(*initialisation de l'opération*)
OP_Purge(
	CTRL_PLC:= CTRL_PLC,
	RESET:= RESET,
	ENABLE_INT:= IN_FE11T AND IN_FE12T AND OP_Test_RP.AR,
	MANUAL:= MANUAL,
	RESTART_ENABLE_IF_OK:= FALSE,
	N_STEP_OP_OK:= 7,
	N_STEP_OP_NOK:=0);

(*appel de l'action de préparation de l'opération*)
OP_Purge.PRL();


(*GRAFCET*)
(* initialisation du grafcet*)
IF 		OP_Purge.Etape = 0
		THEN
				OP_Purge.Etape.0:= TRUE;
(*repositionnement sur étape 0*)
ELSIF	MANUAL OR RESET OR OP_Arret_Pompes.Etape.1
		OR (OP_Isolement.Etape.1 AND NOT OP_Ventilation.Etape.1)
		OR (OP_Pompage_Sec.Etape.1 AND NOT OP_Purge.Etape.6)
		THEN
				OP_Purge.Etape := 0;
				OP_Purge.Etape.0:=TRUE;
(*étape 0-1*)
ELSIF 	OP_Purge.Etape.0
		AND OP_Purge.Marche_OP
		THEN
				OP_Purge.Etape.1:=TRUE;
				OP_Purge.Etape.0:=FALSE;
(*étape 1-2*)
ELSIF	OP_Purge.Etape.1
		AND OP_Pompage_Sec.Etape.0 AND OP_Pompage_Prim.Etape.0 AND OP_Pompage_Proc.Etape.0
		AND OP_Ventilation.Etape.0 AND OP_Isolement.Etape.0
		THEN
				OP_Purge.Etape.2:=TRUE;
				OP_Purge.Etape.1:=FALSE;
(*étape 2-3*)
ELSIF 	OP_Purge.Etape.2
		AND OP_Pompage_Prim.OK AND TH_Vide_Primaire
		THEN
				OP_Purge.Etape.3:=TRUE;
				OP_Purge.Etape.2:=FALSE;
(*étape 3-4*)
ELSIF 	OP_Purge.Etape.3
		AND TIMER_Purge.Q
		THEN
				OP_Purge.Etape.4:=TRUE;
				OP_Purge.Etape.3:=FALSE;
(*étape 3-2*)
ELSIF 	OP_Purge.Etape.3
		AND NOT OP_Pompage_Prim.OK
		THEN
				OP_Purge.Etape.2:=TRUE;
				OP_Purge.Etape.3:=FALSE;
(*étape 4-5*)
ELSIF 	OP_Purge.Etape.4
		AND TH_Atm
		THEN
				OP_Purge.Etape.5:=TRUE;
				OP_Purge.Etape.4:=FALSE;
(*étape 5-2*)
ELSIF 	OP_Purge.Etape.5
		AND (VAR_Iter_Purge < PRM_N_Purge)
		THEN
				OP_Purge.Etape.2:=TRUE;
				OP_Purge.Etape.5:=FALSE;
(*étape 5-6*)
ELSIF 	OP_Purge.Etape.5
		AND (VAR_Iter_Purge >= PRM_N_Purge)
		THEN
				OP_Purge.Etape.6:=TRUE;
				OP_Purge.Etape.5:=FALSE;
(*étape 6-7*)
ELSIF 	OP_Purge.Etape.6
		AND OP_Pompage_Sec.EC
		THEN
				OP_Purge.Etape.7:=TRUE;
				OP_Purge.Etape.6:=FALSE;
END_IF;

(*cloture du traitement de l'opération*)
OP_Purge.POST();
END_ACTION

ACTION ACT_REGEN:
(*OPERATION REGENERATION POMPE CRYOGENIQUE*)
(*isolement pompage et lancement régénération*)

(*initialisation de l'opération*)
OP_Regen(
	CTRL_PLC:= CTRL_PLC,
	RESET:= RESET,
	ENABLE_INT:= OP_Test_RP.AR AND NOT OP_Marche_Pompes.AR,
	MANUAL:= MANUAL,
	RESTART_ENABLE_IF_OK:= FALSE,
	N_STEP_OP_OK:= 6,
	N_STEP_OP_NOK:=0);

(*appel de l'action de préparation de l'opération*)
OP_Regen.PRL();


(*GRAFCET*)
(* initialisation du grafcet*)
IF 		OP_Regen.Etape = 0
		THEN
				OP_Regen.Etape.0:= TRUE;
(*repositionnement sur étape 0*)
ELSIF	MANUAL OR RESET OR OP_Arret_Pompes.Etape.1
		THEN
				OP_Regen.Etape := 0;
				OP_Regen.Etape.0:=TRUE;
(*étape 0-1*)
ELSIF 	OP_Regen.Etape.0
		AND (OP_Regen.Marche_OP OR (FM_REGEN.Q AND NOT MANUAL AND NOT OP_Regen_Part.EC))
		THEN
				OP_Regen.Etape.1:=TRUE;
				OP_Regen.Etape.0:=FALSE;
(*étape 1-2*)
ELSIF	OP_Regen.Etape.1
		THEN
				OP_Regen.Etape.2:=TRUE;
				OP_Regen.Etape.1:=FALSE;
(*étape 2-3*)
ELSIF 	OP_Regen.Etape.2
		AND (OP_Isolement.Etape.4 OR (OP_Pompage_Prim.Etape.0 AND OP_Pompage_Proc.Etape.0 OR OP_Pompage_Sec.Etape.0 OR OP_Purge.Etape.0))
		THEN
				OP_Regen.Etape.3:=TRUE;
				OP_Regen.Etape.2:=FALSE;
(*étape 3-4*)
ELSIF	OP_Regen.Etape.3 AND PS11.STATE_Regen
		THEN
				OP_Regen.Etape.4:=TRUE;
				OP_Regen.Etape.3:=FALSE;
(*étape 4-5*)
ELSIF	OP_Regen.Etape.4 AND NOT PS11.STATE_Regen
		THEN
				OP_Regen.Etape.5:=TRUE;
				OP_Regen.Etape.4:=FALSE;
(*étape 5-6*)
ELSIF	OP_Regen.Etape.5
		AND (OP_Pompage_Sec.OK OR (OP_Marche_Pompes.OK AND (TH_Atm OR NOT OP_Pompage_Sec.ENABLE_INT)))
		THEN
				OP_Regen.Etape.6:=TRUE;
				OP_Regen.Etape.5:=FALSE;
(*étape 6-0*)
ELSIF	OP_Regen.Etape.6
		AND TIMER_etape6_regen.Q
		THEN
				OP_Regen.Etape.0:=TRUE;
				OP_Regen.Etape.6:=FALSE;
END_IF;

(*cloture du traitement de l'opération*)
OP_Regen.POST();
END_ACTION

ACTION ACT_REGEN_PART:
(*OPERATION REGENERATION POMPE CRYOGENIQUE*)
(*isolement pompage et lancement régénération*)

(*initialisation de l'opération*)
OP_Regen_Part(
	CTRL_PLC:= CTRL_PLC,
	RESET:= RESET,
	ENABLE_INT:= OP_Test_RP.AR AND NOT OP_Marche_Pompes.AR,
	MANUAL:= MANUAL,
	RESTART_ENABLE_IF_OK:= FALSE,
	N_STEP_OP_OK:= 6,
	N_STEP_OP_NOK:=0);

(*appel de l'action de préparation de l'opération*)
OP_Regen_Part.PRL();


(*GRAFCET*)
(* initialisation du grafcet*)
IF 		OP_Regen_Part.Etape = 0
		THEN
				OP_Regen_Part.Etape.0:= TRUE;
(*repositionnement sur étape 0*)
ELSIF	MANUAL OR RESET OR OP_Arret_Pompes.Etape.1
		OR OP_Pompage_Sec.Etape.1 OR OP_Pompage_Prim.Etape.1
		THEN
				OP_Regen_Part.Etape := 0;
				OP_Regen_Part.Etape.0:=TRUE;
(*étape 0-1*)
ELSIF 	OP_Regen_Part.Etape.0
		AND OP_Regen_Part.Marche_OP
		THEN
				OP_Regen_Part.Etape.1:=TRUE;
				OP_Regen_Part.Etape.0:=FALSE;
(*étape 1-2*)
ELSIF	OP_Regen_Part.Etape.1
		THEN
				OP_Regen_Part.Etape.2:=TRUE;
				OP_Regen_Part.Etape.1:=FALSE;
(*étape 2-3*)
ELSIF 	OP_Regen_Part.Etape.2
		AND (OP_Isolement.OK
		OR (OP_Pompage_Prim.Etape.0 AND OP_Pompage_Proc.Etape.0 OR OP_Pompage_Sec.Etape.0 OR OP_Purge.Etape.0))
		THEN
				OP_Regen_Part.Etape.3:=TRUE;
				OP_Regen_Part.Etape.2:=FALSE;
(*étape 3-4*)
ELSIF	OP_Regen_Part.Etape.3 AND PS11.STATE_Regen
		THEN
				OP_Regen_Part.Etape.4:=TRUE;
				OP_Regen_Part.Etape.3:=FALSE;
(*étape 4-5*)
ELSIF	OP_Regen_Part.Etape.4
		AND IN_Temp_Etage1 > 300
		THEN
				OP_Regen_Part.Etape.5:=TRUE;
				OP_Regen_Part.Etape.4:=FALSE;
(*étape 5-6*)
ELSIF	OP_Regen_Part.Etape.5
		AND (IN_Temp_Etage1 < PRM_Temp_Post_Purge
			OR TIMER_Post_Purge.Q )
		THEN
				OP_Regen_Part.Etape.6:=TRUE;
				OP_Regen_Part.Etape.5:=FALSE;
(*étape 6-0*)
ELSIF	OP_Regen_Part.Etape.6
		AND TIMER_etape6_regen.Q
		THEN
				OP_Regen_Part.Etape.0:=TRUE;
				OP_Regen_Part.Etape.6:=FALSE;
END_IF;

(*cloture du traitement de l'opération*)
OP_Regen_Part.POST();
END_ACTION

ACTION ACT_TEST_RP:
(*OPERATION TEST REMONTEE PRESSION*)

OP_TEST_RP(
	CTRL_PLC:= CTRL_PLC,
	RESET:= RESET,
	MANUAL:=MANUAL ,
	ENABLE_INT := OP_Pompage_Sec.OK AND OP_Purge.AR AND OP_Regen.AR AND OP_Regen_Part.AR,
	RESTART_ENABLE_IF_OK:=TRUE ,
	N_STEP_OP_OK:= 8,
	N_STEP_OP_NOK:=0 );

(*appel de l'action de préparation de l'opération*)
OP_TEST_RP.PRL();

(*GRAFCET*)
(* initialisation du grafcet*)
IF 		OP_TEST_RP.ETAPE = 0
		THEN
				OP_TEST_RP.ETAPE.0 := TRUE;
(*repositionnement sur étape 0*)
ELSIF 	RESET OR MANUAL OR (OP_Isolement.Etape.1 AND NOT OP_Test_RP.Etape.3)
			OR (OP_Pompage_Sec.Etape.1 AND OP_Test_RP.Etape.3) OR CO_Stop_Test_RP
			OR OP_Arret_Pompes.Etape.1 OR OP_Isolement.ON_AUTO_EXT OR OP_Isolement.ON_AUTO_INT
		THEN
				OP_TEST_RP.ETAPE := 0;
				OP_TEST_RP.ETAPE.0:=TRUE;
(*étape 0-1*)
ELSIF 	OP_TEST_RP.ETAPE.0 AND OP_TEST_RP.MARCHE_OP
		THEN
				OP_TEST_RP.ETAPE.1:=TRUE;
				OP_TEST_RP.ETAPE.0:=FALSE;
(*étape 1-2*)
ELSIF 	OP_TEST_RP.ETAPE.1
		THEN
				OP_TEST_RP.ETAPE.2:=TRUE;
				OP_TEST_RP.ETAPE.1:=FALSE;
(*étape 2-3*)
ELSIF 	OP_TEST_RP.ETAPE.2
		AND OP_Pompage_Sec.ok AND TH_Test_RP
		THEN
				OP_TEST_RP.ETAPE.3:=TRUE;
				OP_TEST_RP.ETAPE.2:=FALSE;
(*étape 3-4*)
ELSIF 	OP_TEST_RP.ETAPE.3
		AND OP_Isolement.OK
		THEN
				OP_TEST_RP.ETAPE.4:=TRUE;
				OP_TEST_RP.ETAPE.3:=FALSE;
(*étape 4-5*)
ELSIF 	OP_TEST_RP.ETAPE.4
		AND TIMER_attente_test.Q
		THEN
				OP_TEST_RP.ETAPE.5:=TRUE;
				OP_TEST_RP.ETAPE.4:=FALSE;
(*étape 5-6*)
ELSIF 	OP_TEST_RP.ETAPE.5
		THEN
				OP_TEST_RP.ETAPE.6:=TRUE;
				OP_TEST_RP.ETAPE.5:=FALSE;
(*étape 6-7*)
ELSIF 	OP_TEST_RP.ETAPE.6
		THEN
				OP_TEST_RP.ETAPE.7:=TRUE;
				OP_TEST_RP.ETAPE.6:=FALSE;
(*étape 7-8*)
ELSIF 	OP_TEST_RP.ETAPE.7
		AND OP_Pompage_Sec.OK
		THEN
				OP_TEST_RP.ETAPE.8:=TRUE;
				OP_TEST_RP.ETAPE.7:=FALSE;
(*étape 8-1*)
ELSIF 	OP_TEST_RP.ETAPE.8 AND OP_TEST_RP.MARCHE_OP
		THEN
				OP_TEST_RP.ETAPE.1:=TRUE;
				OP_TEST_RP.ETAPE.8:=FALSE;
END_IF
(*cloture du traitement de l'opération*)
OP_TEST_RP.POST();
CO_Stop_Test_RP	:=	FALSE;
END_ACTION

ACTION ACT_VENTILATION:
(*OPERATION VENTILATION*)


(*initialisation de l'opération*)
OP_Ventilation(
	CTRL_PLC:= CTRL_PLC,
	RESET:= RESET,
	ENABLE_INT:=OP_Purge.Etape.0,
	MANUAL:= MANUAL,
	ON_AUTO_INT:= FALSE ,
	RESTART_ENABLE_IF_OK:= FALSE,
	N_STEP_OP_OK:= 8,
	N_STEP_OP_NOK:=0);

(*appel de l'action de préparation de l'opération*)
OP_Ventilation.PRL();


(*GRAFCET*)
(* initialisation du grafcet*)
IF 		OP_Ventilation.Etape = 0
		THEN
				OP_Ventilation.Etape.0:= TRUE;
(*repositionnement sur étape 0*)
ELSIF	MANUAL OR RESET OR (OP_isolement.Etape.1 AND NOT  OP_ventilation.Etape.1)
		OR OP_Pompage_sec.Etape.1 OR Op_Pompage_Prim.Etape.1
		OR OP_Pompage_Proc.Etape.1 OR OP_Purge.Etape.1
		THEN
				OP_Ventilation.Etape := 0;
				OP_Ventilation.Etape.0:=TRUE;
(*étape 0-1*)
ELSIF 	OP_Ventilation.Etape.0
		 AND (OP_Ventilation.Marche_OP OR OP_Purge.Etape.4)
		THEN
				OP_Ventilation.Etape.1:=TRUE;
				OP_Ventilation.Etape.0:=FALSE;
(*étape 1-9*)
ELSIF	OP_Ventilation.Etape.1
		AND OP_isolement.OK THEN
				OP_Ventilation.Etape.9:=TRUE;
				OP_Ventilation.Etape.1:=FALSE;
(*étape 9-2*)
ELSIF	OP_Ventilation.Etape.9
		AND OP_isolement.Etape.0 THEN
				OP_Ventilation.Etape.2:=TRUE;
				OP_Ventilation.Etape.9:=FALSE;
(*étape 2-3*)
ELSIF 	OP_Ventilation.Etape.2 AND  I_Prep_Ventil_Ok  THEN
				OP_Ventilation.Etape.3:=TRUE;
				OP_Ventilation.Etape.2:=FALSE;
(*étape 3-4*)
ELSIF	OP_Ventilation.Etape.3
		AND  I_Stop_Mesure_OK   THEN
				OP_Ventilation.Etape.4:=TRUE;
				OP_Ventilation.Etape.3:=FALSE;
(*étape 4-5*)
ELSIF	OP_Ventilation.Etape.4
		THEN
				OP_Ventilation.Etape.5:=TRUE;
				OP_Ventilation.Etape.4:=FALSE;
(*étape 5-6*)
ELSIF 	OP_Ventilation.Etape.5
		AND (TH_atm OR I_Fin_Ventil OR NOT IN_FE11T OR NOT IN_FE12T )
		THEN
				OP_Ventilation.Etape.6:=TRUE;
				OP_Ventilation.Etape.5:=FALSE;
(*étape 6-7*)
ELSIF 	OP_Ventilation.Etape.6
		AND (TIMER_SurVentilation_enc.Q OR I_Fin_Ventil OR NOT IN_FE11T OR NOT IN_FE12T)
		THEN
				OP_Ventilation.Etape.7:=TRUE;
				OP_Ventilation.Etape.6:=FALSE;
(*étape 7-8*)
ELSIF 	OP_Ventilation.Etape.7
		AND VH11.STATE_Off THEN
				OP_Ventilation.Etape.8:=TRUE;
				OP_Ventilation.Etape.7:=FALSE;
END_IF;

(*cloture du traitement de l'opération*)
OP_Ventilation.POST();
END_ACTION

ACTION POST:
VAR_Reset_Sortie := 	NOT MANUAL AND OP_Arret_Pompes.Etape.0 AND OP_Isolement.Etape.0 AND OP_Marche_Pompes.Etape.0
					AND OP_Pompage_Prim.Etape.0 AND OP_Pompage_Proc.Etape.0 AND OP_Pompage_Sec.Etape.0
					AND OP_Ventilation.Etape.0 AND OP_Purge.Etape.0 AND OP_Regen.Etape.0 AND OP_Regen_Part.Etape.0;




(*****************************************)
(*       pompe primaire PP11             *)
(*****************************************)
IF (OP_MARCHE_POMPES.ETAPE.2 AND CONF_Pompage_interjoint)
	OR OP_Pompage_Prim.Etape.3
	OR PS11.STATE_Regen AND NOT RESET
	THEN
		PP11.CO_On 	:= 	TRUE;
ELSIF RESET OR (VAR_Reset_Sortie AND NOT PS11.STATE_Regen)
    OR (OP_Pompage_Sec.Etape.5 AND PR11.STATE_Off AND NOT CONF_Pompage_interjoint)
	OR (OP_Isolement.Etape.3 AND PR11.STATE_Off AND NOT PS11.STATE_Regen  AND NOT CONF_Pompage_interjoint)
	OR OP_Arret_Pompes.Etape.6 AND PR11.STATE_Off AND VP11.STATE_Off
	THEN
		PP11.CO_On	:= 	FALSE;
END_IF;

(*****************************************)
(*       pompe primaire PR11             *)
(*****************************************)
TIMER_Arret_Roots.IN := (OP_Pompage_Sec.OK
						OR (OP_Pompage_Prim.AR AND VP11.STATE_Off AND NOT PS11.STATE_Regen)) AND CONF_Pompage_interjoint;
TIMER_Arret_Roots.PT := T#2M;
TIMER_Arret_Roots();

IF (OP_Pompage_Prim.Etape.3 AND PP11.STATE_On)
	OR (PS11.STATE_Regen AND PP11.STATE_On AND NOT RESET) THEN
		PR11.CO_On 	:= 	TRUE;
ELSIF RESET OR VAR_Reset_Sortie
    OR TIMER_Arret_Roots.Q
	OR OP_Arret_Pompes.Etape.3 
	OR (OP_Isolement.Etape.3 AND NOT PS11.STATE_Regen AND NOT CONF_Pompage_interjoint)
	OR (OP_Pompage_Sec.Etape.5 AND NOT CONF_Pompage_interjoint)
	THEN
		PR11.CO_On	:= 	FALSE;
END_IF;

(*****************************************)
(* 		pompe cryo PS11		   *)
(*****************************************)
IF  OP_Marche_Pompes.Etape.4  THEN
	PS11.CO_On 	:= 	TRUE;
ELSIF RESET  (*OR VAR_Reset_Sortie TODOLN*)  OR OP_Arret_Pompes.Etape.3 THEN
	PS11.CO_On	:= 	FALSE;
	PS11.CO_Regen := FALSE;
END_IF;
IF OP_Regen.Etape.3 OR OP_Regen_Part.Etape.3 THEN
	PS11.CO_Regen	:=	TRUE;
ELSIF OP_Regen.Etape.4 OR OP_Regen_Part.Etape.4 THEN
	PS11.CO_Regen	:=	FALSE;
ELSIF MANUAL THEN
	PS11.CO_On		:=	PS11.VAR_On;
END_IF;

(*****************************************)
(* 		vanne VP11    		   *)
(*****************************************)
IF OP_Pompage_Prim.Etape.4   THEN
		VP11.CO_On 		:= 	TRUE;
ELSIF RESET OR VAR_Reset_Sortie OR OP_Pompage_Sec.Etape.4  OR OP_Isolement.Etape.2 THEN
		VP11.CO_On		:= 	FALSE;
END_IF;


(******************************************)
(*		Vanne  VH11		              *)
(******************************************)
IF   OP_VENTILATION.Etape.5 OR OP_Ventilation.Etape.6 THEN
			VH11.CO_On 	:= 	TRUE;
ELSIF RESET OR  VAR_Reset_Sortie OR OP_Pompage_Prim.Etape.1 OR
	   OP_Pompage_Sec.Etape.2 OR   OP_Isolement.Etape.2 OR OP_Ventilation.Etape.7
	   THEN
			VH11.CO_On	:= 	FALSE;
END_IF;

(******************************************)
(*                  Vanne  VS11                       *)
(******************************************)
IF OP_Pompage_Sec.Etape.6   THEN
		VS11.CO_On 	:= 	TRUE;
		VS11.CO_Lam:=	FALSE;
ELSIF OP_Pompage_Proc.Etape.2  THEN
		VS11.CO_On 	:= 	FALSE;
		VS11.CO_Lam:=	TRUE;
ELSIF VAR_Reset_Sortie OR RESET
	   OR OP_Pompage_Prim.Etape.1   OR OP_Isolement.Etape.2 THEN
		VS11.CO_On	:= 	FALSE;
		VS11.CO_Lam:=	FALSE;
END_IF;


(******************************************)
(*                 Vanne  VINT                    *)
(******************************************)
VINT.CO_On 	:= 	G7_Bal_Int.Etape.6 OR G7_Bal_Int.Etape.7 OR G7_Bal_Int.Etape.11 OR G7_Bal_Int.Etape.12;


(******************************************)
(*                 Vanne  VN2PP11                *)
(******************************************)
VN2PP11.CO_On 	:= 	G7_Bal_Int.Etape.3 OR G7_Bal_Int.Etape.4 OR G7_Bal_Int.Etape.15 OR G7_Bal_Int.Etape.16 OR G7_Bal_Int.Etape.24;



(***********************************************)
(*                Demande diverse              *)
(***********************************************)

(*demande de préparation avant ventilation*)
RQ_Prep_Ventil_Enc 	:= OP_VENTILATION.Etape.2;

(*Demande d'arrêt de la mesure avant ventilation enceinte*)
RQ_Stop_Mesure_Enc := Op_Ventilation.Etape.3 OR Op_Ventilation.Etape.4 OR Op_Ventilation.Etape.5 ;

(*Tempo de surventilation enceinte*)
TIMER_SurVentilation_Enc	(
					PT:=PRM_Tim_SurVentil_E,
					IN:=OP_VENTILATION.Etape.6 AND TH_Atm
					);

(*Temporisation d'arrêt pompe primaire*)
TIMER_Arret_PP11(
					PT:=PRM_Tim_Arret_PP11,
					IN:=OP_Arret_Pompes.Etape.3,
				);

(*Tempo de purge*)
TIMER_Purge (
					PT:=PRM_Tim_Purge,
					IN:=OP_Purge.Etape.3
					);

(*Compteur d'itération purge*)
IF		OP_Purge.Etape.0 THEN
	VAR_Iter_Purge	:=	0;
ELSIF	OP_Purge.Etape.5 THEN
	VAR_Iter_Purge	:=	VAR_Iter_Purge + 1;
END_IF

(*timer de prep ventil*)
TIM_Prep_ventil.PT := PRM_Tim_Prep_Ventil;
TIM_Prep_ventil.IN := OP_Ventilation.Etape.2;
TIM_Prep_ventil();


(*Tempo de retard à l'ouverture de la vanne interjoint*)
IF G7_Bal_Int.etape.4 THEN
	TIMER_BalInt.PT	:=	PRM_Tim_Bal_BalInt;
ELSIF G7_Bal_Int.Etape.7 THEN
	TIMER_BalInt.PT	:=	PRM_Tim_Int_BalInt;
ELSIF G7_Bal_Int.Etape.16 THEN
	TIMER_BalInt.PT	:=	PRM_Tim_FinBal;
END_IF
TIMER_BalInt(IN:=G7_Bal_Int.etape.4 OR G7_Bal_Int.etape.7 OR G7_Bal_Int.etape.16);


(*timer de post purge en regen partielle*)
TIMER_Post_Purge.PT			:=	PRM_Tim_Post_Purge;
TIMER_Post_Purge.IN			:=	OP_Regen_Part.Etape.5;
TIMER_Post_Purge();

TIMER_etape6_regen.PT		:=	T#500ms;
TIMER_etape6_regen.IN		:=	OP_Regen.Etape.6 OR OP_Regen_Part.Etape.6;
TIMER_etape6_regen();

(***************** test de remontée de pression*************************)
TIMER_attente_test		(
					PT:=PRM_Tim_test,
					IN:=OP_Test_RP.Etape.4
					);
(*Mémorisation des pressions lors du test et calcul de l'indicateur*)
IF FM_etape4.Q THEN
	VAR_Mem_Pression_deb := IN_Pressure_RP;
END_IF;
IF OP_Test_RP.Etape.5 THEN
	VAR_Mem_Pression_fin := IN_Pressure_RP;
END_IF;
(*Indicateur final faisant intervenir le volume ATTENTION : FORMULE MEMO SANS DOUTE FAUSSE*)
IF OP_Test_RP.Etape.6 THEN
	VAR_indicateur_test := (VAR_Mem_Pression_fin - VAR_Mem_Pression_deb) * CONF_volume_enceinte / TIME_TO_REAL(PRM_Tim_Test) * 1000;
END_IF;

EV_Test_RP.CONDITION	:=	OP_Test_RP.Etape.7;
EV_Test_RP.VAL1			:=	CONCAT(REAL_TO_STRING(VAR_indicateur_test),' mbar.L/s');
EV_Test_RP();


(*****************************************************)
(* APPEL DES FONCTIONS COMPOSANTS*)
(*****************************************************)

(*Vanne de pompage primaire enceinte*)
VP11(
	RESET:= RESET,
	MANUAL:= MANUAL,
	EN_On_INT:=  PP11.STATE_On AND PR11.STATE_On AND VH11.STATE_Off AND VS11.STATE_Off AND IN_FE11T AND IN_FE12T AND NOT PS11.STATE_Regen,
	EN_Off_INT:= TRUE
	);

(*Vanne pompage secondaire enceinte*)
VS11(
	RESET:= RESET,
	MANUAL:= MANUAL,
	EN_On_INT:= (PS11.STATE_Ok
				AND VP11.STATE_Off AND VH11.STATE_Off)
				AND TH_RP_Enc,
	EN_Off_INT:= TRUE
	);

(*Vanne ventilation enceinte*)
VH11(
	RESET:= RESET,
	MANUAL:= MANUAL,
	EN_On_INT:= VP11.STATE_Off  AND  VS11.STATE_Off,
	EN_Off_INT:= TRUE
	);

(*Vanne interjoint*)
VINT(
	RESET:= RESET,
	MANUAL:= MANUAL,
	EN_On_INT:= PP11.STATE_On AND NOT PS11.STATE_Regen AND VN2PP11.STATE_Off,
	EN_Off_INT:= TRUE
	);
	
(*Vanne balayage pompe primaire*)
VN2PP11(
	RESET:= RESET,
	MANUAL:= MANUAL,
	EN_On_INT:= NOT PS11.STATE_Regen AND VINT.STATE_Off AND VP11.STATE_Off,
	EN_Off_INT:= TRUE
	);

(*Pompe primaire PP11*)
PP11(
	RESET:= 	RESET,
	MANUAL:= 	MANUAL AND NOT PS11.STATE_Regen,
	EN_On_INT:= TRUE,
	EN_Off_INT:= (PR11.STATE_Off AND VP11.STATE_Off AND NOT PS11.STATE_Regen) OR VAR_Reset_sortie
	);
	
(*Pompe roots PR11*)
PR11(
	RESET:= 	RESET,
	MANUAL:= 	MANUAL,
	EN_On_INT:= PP11.STATE_On,
	EN_Off_INT:= (VP11.STATE_Off AND NOT PS11.STATE_Regen) OR VAR_Reset_sortie
	);

(*Pompe cryo PS11*)
PS11(
	RESET:= RESET,
	MANUAL:= MANUAL,
	EN_On_INT:= TRUE ,
	EN_Off_INT:= VS11.STATE_Off OR VAR_Reset_Sortie,
	EN_Regen_INT:= VS11.STATE_Off
	);


(*******************************************)
(* GESTION DES DEFAUTS 	     *)
(*******************************************)


(*Défaut d'obtention du seuil de basculement en pompage secondaire*)
DEF_PPRIM			(
					Condition:=	(OP_Pompage_Prim.Etape.5 AND OP_Pompage_Sec.Etape.3) AND (DEF_PPRIM.DELAY<>T#0ms)

					);
DEF_TGF				(
					Condition:= 	(OP_Pompage_Prim.Etape.5 OR OP_pompage_prim.Etape.4) AND OP_Pompage_sec.Etape.3
								AND	(DEF_TGF.DELAY<>T#0ms) AND NOT TH_Grosse_Fuite
					);

(*Défaut de remontée de pression dans l'enceinte pendant le pompage secondaire*)
(* validation ok - SP *)
DEF_RP_enc			(
					Condition:=	NOT VS11.STATE_Off AND NOT TH_RP_Enc AND NOT RESET
					);

(*Défaut de ventilation*)
DEF_Vent			(
					Condition:=	(OP_ventilation.Etape.4 OR Op_ventilation.Etape.5 OR op_ventilation.Etape.6) AND (DEF_Vent.DELAY <> T#0ms)
					);
END_ACTION

ACTION PRL:
(*vérification pour empécher la division par 0*)
IF TIME_TO_REAL(PRM_Tim_test) = 0 THEN
	PRM_Tim_test := T#1s;
END_IF
FM_etape4(clk := OP_Test_RP.Etape.4);

IdXML							:=	'2';
TagXML							:=	0;

OP_Marche_Pompes.IdXML			:= 	'1';
OP_Marche_Pompes.TagXML			:=	1;

OP_Arret_Pompes.IdXML			:= 	'1';
OP_Arret_Pompes.TagXML			:= 	2;

OP_Isolement.IdXML				:= 	'1';
OP_Isolement.TagXML				:= 	3;

OP_Ventilation.IdXML			:= 	'1';
OP_Ventilation.TagXML			:= 	4;

OP_Pompage_Prim.IdXML			:=	'1';
OP_Pompage_Prim.TagXML			:=	6;

OP_Pompage_Sec.IdXML			:=	'1';
OP_Pompage_Sec.TagXML			:=	5;

OP_Pompage_Proc.IdXML			:=	'1';
OP_Pompage_Proc.TagXML			:=	7;

OP_Purge.IdXML					:=	'1';
OP_Purge.TagXML					:=	8;

OP_Regen.IdXML					:=	'1';
OP_Regen.TagXML					:=	9;

OP_Test_RP.IdXML				:=	'1';
OP_Test_RP.TagXML				:=	10;


DEF_PPrim.IdXML					:= '1';
DEF_PPrim.TagXML				:= 1;
DEF_Vent.IdXML					:= '1';
DEF_Vent.TagXML					:= 2;
DEF_RP_enc.IdXML				:= '1';
DEF_RP_enc.TagXML				:= 3;
DEF_TGF.IdXML					:= '1';
DEF_TGF.TagXML					:= 4;
	
EV_Test_RP.IdXML				:=	'1';
EV_Test_RP.TagXML				:=	14;
EV_Test_RP.Groupe				:=	3;

PP11.IdXML					:=	'1';
PP11.TagXML					:=	7;

PR11.IdXML					:=	'1';
PR11.TagXML					:=	10;

PS11.IdXML					:=	'1';
PS11.TagXML					:=	9;

VP11.IdXML					:=	'1';
VP11.TagXML					:=	2;
VP11.DEF_On.IdXML			:=	'3';
VP11.DEF_On.TagXML			:=	2;
VP11.DEF_Off.IdXML			:=	'3';
VP11.DEF_Off.TagXML			:=	4;
VP11.DEF_Sensor.IdXML		:=	'3';
VP11.DEF_Sensor.TagXML		:=	13;
VP11.DEF_On_Imposs.IdXML	:=	'3';
VP11.DEF_On_Imposs.TagXML	:=	6;
VP11.DEF_Off_Imposs.IdXML	:=	'3';
VP11.DEF_Off_Imposs.TagXML	:=	9;
VP11.DEF_Off_auto.IdXML		:=	'3';
VP11.DEF_Off_auto.TagXML	:=	11;

VH11.IdXML					:=	'1';
VH11.TagXML					:=	4;
VH11.DEF_On.IdXML			:=	'3';
VH11.DEF_On.TagXML			:=	2;
VH11.DEF_Off.IdXML			:=	'3';
VH11.DEF_Off.TagXML			:=	4;
VH11.DEF_Sensor.IdXML		:=	'3';
VH11.DEF_Sensor.TagXML		:=	13;
VH11.DEF_On_Imposs.IdXML	:=	'3';
VH11.DEF_On_Imposs.TagXML	:=	6;
VH11.DEF_Off_Imposs.IdXML	:=	'3';
VH11.DEF_Off_Imposs.TagXML	:=	9;
VH11.DEF_Off_auto.IdXML		:=	'3';
VH11.DEF_Off_auto.TagXML	:=	11;

VS11.IdXML					:=	'1';
VS11.TagXML					:=	3;

VINT.IdXML					:=	'1';
VINT.TagXML					:=	1;
VINT.DEF_On.IdXML			:=	'3';
VINT.DEF_On.TagXML			:=	2;
VINT.DEF_Off.IdXML			:=	'3';
VINT.DEF_Off.TagXML			:=	4;
VINT.DEF_Sensor.IdXML		:=	'3';
VINT.DEF_Sensor.TagXML		:=	13;
VINT.DEF_On_Imposs.IdXML	:=	'3';
VINT.DEF_On_Imposs.TagXML	:=	6;
VINT.DEF_Off_Imposs.IdXML	:=	'3';
VINT.DEF_Off_Imposs.TagXML	:=	9;
VINT.DEF_Off_auto.IdXML		:=	'3';
VINT.DEF_Off_auto.TagXML	:=	11;


VN2PP11.IdXML					:=	'1';
VN2PP11.TagXML					:=	1;
VN2PP11.DEF_On.IdXML			:=	'3';
VN2PP11.DEF_On.TagXML			:=	2;
VN2PP11.DEF_Off.IdXML			:=	'3';
VN2PP11.DEF_Off.TagXML			:=	4;
VN2PP11.DEF_Sensor.IdXML		:=	'3';
VN2PP11.DEF_Sensor.TagXML		:=	13;
VN2PP11.DEF_On_Imposs.IdXML		:=	'3';
VN2PP11.DEF_On_Imposs.TagXML	:=	6;
VN2PP11.DEF_Off_Imposs.IdXML	:=	'3';
VN2PP11.DEF_Off_Imposs.TagXML	:=	9;
VN2PP11.DEF_Off_auto.IdXML		:=	'3';
VN2PP11.DEF_Off_auto.TagXML		:=	11;

(* Gestion FM et FD régénération*)
FM_REGEN(CLK:=PS11.STATE_Regen);
FD_REGEN(CLK:=PS11.STATE_Regen);
END_ACTION

END_FUNCTION_BLOCK

// ---- POUs/Composant/VANNES/BLOCK_VVAT_3P.TcPOU
FUNCTION_BLOCK BLOCK_VVAT_3P

(* Gestion d'une vanne 3 positions VAT*)

(****************historique des versions*****************************)

(* Version 1-0 - SP - VERSION INIITIALE 6844 DP650 N35*)
(* Version 2-0 - LDS - 5236 EVA900 N1 - inversion des sorti V11 et V12*)
(*************************************************************************)


VAR_INPUT
	I_PARAM_SYSTEM_OK:		BOOL;
(*paramètre standard*)
	RESET:   				BOOL; 												(*Condition RAZ actionneur*)
	MANUAL:  				BOOL;												(*Mode manuel*)

	(*Entité*)
	IsComponent:			BOOL;			(*entité : composant*)
	IdXML:					STRING;			(*nom entité : identifiant pour recherche dans dico*)
	TagXML:					UINT;			(*nom entité : identifiant pour recherche dans dico*)
	IdParent:				STRING;			(*MNEMO de l'appelant*)
	MNEMO:					STRING;			(*MNEMO de l'entité*)

(*entrée externe*)
	IN_OFF:						BOOL; (* ~ (OPC : 1 : available for OPC-clients) *)		(*E.TOR vanne fermée*)
	IN_ON:						BOOL; (* ~ (OPC : 1 : available for OPC-clients) *)		(*E.TOR vanne ouverte*)
	IN_LAM:						BOOL; (* ~ (OPC : 1 : available for OPC-clients) *)		(*E.TOR vanne en position de laminage*)

(*défaut du bloc*)
	DEF_On:  					PRCDEF; 									(*00 - Défaut d'ouverture de la vanne*)
	DEF_Off:   					PRCDEF; 									(*01 - Défaut de fermeture de la vanne*)
	DEF_Sensor:  				PRCDEF; 									(*02 - Défaut d'incohérence des capteurs de la vanne*)
	DEF_Lam:					PRCDEF;										(*03 - Défaut de positionnement en position de laminage*)
	DEF_On_Imposs:				PRCDEF;										(*04 - Défaut d'ouverture ou de mise en laminage non autorisée en mode automatique*)
	DEF_Off_Imposs:				PRCDEF;										(*05 - Défaut de fermeture non autorisée en mode automatique*)
	DEF_Off_auto:				PRCDEF;										(*06 - Défaut de fermeture automatique de la vanne*)

(*parametre de pilotage en entrée*)
	CO_On:   					BOOL; 										(*Ordre mode automatique ouverture*)
	CO_Lam:						BOOL;										(*Ordre mode automatique laminage*)
	EN_On_INT:   				BOOL;										(*Condition d'autorisation d'ouverture ou de laminage donnée par le bloc qui instancie le bloc actuator*)
	EN_Off_INT:  				BOOL; 										(*Condition d'autorisation de fermeture donnée par le bloc qui instacie le bloc actuator*)
	EN_On_EXT:					BOOL:=TRUE;									(*condition d'autorisation d'ouverture ou de laminage externe*)
	EN_Off_EXT:					BOOL:=TRUE;									(*condition d'autorisation de fermeture externe*)
END_VAR

VAR_INPUT PERSISTENT
(*parametre de configuration constructeur*)
(*les parametres suivants dépendent de la configuration de la machine*)
	CONF_DI_Off:   				BOOL:=FALSE;			(*option de presence d'un capteur desactivation ok*)
	CONF_DI_On:  				BOOL:=FALSE;			(*option de presence d'un capteur activation ok*)
	CONF_DI_Lam:				BOOL:=FALSE;			(*option de présence d'un capteur de position laminage *)
	CONF_Tim_Valid_On:  		TIME:=T#100MS; 			(*Temps validation de la position ouverte *)
	CONF_Tim_Valid_Off:   		TIME:=T#100ms; 			(*Temps validation de la position fermée *)
	CONF_Tim_Valid_Lam:			TIME:=T#100MS;			(*Temps de validation de la position laminage*)
	CONF_EN_On:					USINT:=0;				(*définit la réaction du système en cas de perte des conditions d'autorisation d'activation EN_On*)
														(* 0 = désactivation automatique  en cas de perte des conditions d'autorisation d'activation uniquement en manuel*)
														(* 1 = désactivation automatique en cas de perte des conditions d'autorisation d'activation en auto et en manuel*)
														(* 2 = Pas de déscativation automatique*)

END_VAR

VAR_OUTPUT
	OUT_V11:					BOOL;	(* ~ (OPC : 1 : available for OPC-clients) *)		(*SORTIE OUVERTURE VANNE*)
	OUT_V12:					BOOL; 	(* ~ (OPC : 1 : available for OPC-clients) *)		(*SORTIE MISE EN LAMINAGE*)
	STATE_On:	   				BOOL; 	(* ~ (OPC : 1 : available for OPC-clients) *)		(*Indicateur ouverture ok*)
	STATE_Off:  				BOOL; 	(* ~ (OPC : 1 : available for OPC-clients) *)		(*Indicateur fermeture ok*)
	STATE_Nok:					BOOL;	(* ~ (OPC : 1 : available for OPC-clients) *)		(*Indicateur défaut sur la vanne*)
	STATE_Lam:					BOOL;	(* ~ (OPC : 1 : available for OPC-clients) *)		(*Indicateur laminage ok*)
	AUTOR_On_IHM:				BOOL; 	(* ~ (OPC : 1 : available for OPC-clients) *)		(*etat ouverture autorisée depuis la supervision en mode manuel*)
	AUTOR_Off_IHM:				BOOL; 	(* ~ (OPC : 1 : available for OPC-clients) *)		(*etat fermeture autorisée depuis la supervision en mode manuel*)
	AUTOR_Lam_IHM:				BOOL;	(* ~ (OPC : 1 : available for OPC-clients) *)		(*etat laminage autorisée depuis la supervision en mode manuel*)
	AUTOR_On_PLC:				BOOL;											(*etat ouverture autorisée depuis l'automate*)
	AUTOR_Off_PLC:				BOOL;											(*etat fermeture autorisée depuis l'automate*)
END_VAR


VAR
	TIMER_Valid_On:				TON;
	TIMER_Valid_Off:			TON;
	TIMER_Valid_Lam:			TON;

	M_On:  						BOOL; 	(* ~ (OPC : 1 : available for OPC-clients) *)		(*Ordre mode manuel ouverture de la vanne*)
	M_Off:   					BOOL; 	(* ~ (OPC : 1 : available for OPC-clients) *)		(*Ordre mode manuel fermeture de la vanne*)
	M_Lam:   					BOOL; 	(* ~ (OPC : 1 : available for OPC-clients) *)		(*Ordre mode manuel de mise en position laminage*)
	RCP_M_On:   				BOOL;
	RCP_M_Off:  				BOOL;
	RCP_M_Lam:					BOOL;
	VAR_On:						BOOL;											(*bit intermédiaire de demande d'ouverture de la vanne*)
	VAR_Lam:					BOOL;											(*bit intermédiaire de demande de mise en laminage de la vanne*)

	bTest:						BOOL;

END_VAR

VAR_EXTERNAL
	MANUAL_SAFETY_OFF:			BOOL;											(*desactive les sécurités en mode manuel*)
END_VAR

DEF_Off_Auto.IdXml				:=	'3';
DEF_Off_Auto.TagXml				:=	11;

DEF_On_imposs.IdXml				:=	'3';
DEF_On_imposs.TagXml			:=	7;

DEF_Off_imposs.IdXml			:=	'3';
DEF_Off_imposs.TagXml			:=	9;

DEF_On.IdXml					:=	'3';
DEF_On.TagXml					:=	2;

DEF_Off.IdXml					:=	'3';
DEF_Off.TagXml					:=	4;

DEF_Sensor.IdXML				:=	'3';
DEF_Sensor.TagXML 				:=	13;

DEF_Lam.IdXML					:=	'3';
DEF_Lam.TagXML 					:=	18;

(* Réception des ordres en mode manuel*)
RCP_M_On 			:=	M_On;
RCP_M_Off			:=	M_Off;
RCP_M_Lam			:=	M_Lam;
(*Autorisation*)
AUTOR_On_IHM		:= 	MANUAL AND ((EN_On_INT AND EN_On_EXT)
						OR MANUAL_SAFETY_OFF) AND NOT RESET AND NOT VAR_On;
AUTOR_Off_IHM		:= 	MANUAL AND ((EN_Off_INT AND EN_Off_EXT)  OR
						MANUAL_SAFETY_OFF) AND NOT RESET AND  (VAR_On OR VAR_Lam);
AUTOR_Lam_IHM		:=	MANUAL AND ((EN_On_INT AND EN_On_EXT)
						OR MANUAL_SAFETY_OFF) AND NOT RESET AND NOT VAR_Lam;
AUTOR_On_PLC		:=	NOT MANUAL AND (EN_On_INT AND EN_On_EXT)
						AND NOT RESET;
AUTOR_Off_PLC		:= 	NOT MANUAL AND (EN_Off_INT AND EN_Off_EXT)
						AND NOT RESET;

(*defaut ouverture ou laminage impossible en mode automatique*)
DEF_On_Imposs.CONDITION:=	(CO_On OR CO_Lam) AND NOT AUTOR_On_PLC
							AND NOT MANUAL AND NOT RESET;
DEF_On_Imposs.DELAY := T#0ms;
DEF_On_Imposs();
(*Defaut fermeture impossible en mode automatique*)
DEF_Off_Imposs.CONDITION:=	NOT CO_On AND NOT CO_Lam AND NOT AUTOR_Off_PLC
							AND NOT MANUAL AND NOT RESET AND (VAR_Lam OR VAR_On);
DEF_Off_Imposs.DELAY := T#0ms;
DEF_Off_Imposs();

(*defaut de fermeture automatique de la vanne*)
DEF_Off_Auto.CONDITION :=             (NOT EN_On_INT OR NOT EN_On_EXT) AND  (VAR_On OR VAR_Lam)
								 AND ((CONF_En_ON=1) OR ((CONF_EN_On=0) AND MANUAL)) AND NOT RESET;
DEF_Off_auto.DELAY:=T#0ms;
DEF_Off_Auto();

(*gestion des sorties*)
IF 		(RCP_M_On AND AUTOR_On_IHM) OR
		(CO_On AND AUTOR_On_PLC) THEN
			VAR_On		:= 	TRUE;
			VAR_Lam	:= 	FALSE;
ELSIF 	(RCP_M_Lam AND AUTOR_Lam_IHM) OR
	    	(CO_Lam AND AUTOR_On_PLC) THEN
			VAR_On		:=	FALSE;
			VAR_LAm	:=	TRUE;
ELSIF 	RESET  OR DEF_Off_Auto.DEF OR
		(RCP_M_Off AND AUTOR_Off_IHM) OR
	    	((NOT CO_Lam AND NOT CO_On) AND AUTOR_Off_PLC) THEN
			VAR_On		:= 	FALSE;
			VAR_Lam	:=	FALSE;
END_IF;

IF DEF_Off_auto.DEF THEN
	bTest:= TRUE;
END_IF


OUT_V11		:=	VAR_On OR VAR_Lam;
OUT_V12		:=	VAR_On;

(*indicateur actionneur activé STATE_ON*)
TIMER_Valid_On.IN	:=	((VAR_ON AND NOT CONF_DI_On AND (NOT CONF_DI_OFF OR NOT IN_Off) AND ( NOT CONF_DI_Lam OR NOT IN_Lam)) OR
						(IN_ON AND CONF_DI_On)) AND NOT DEF_SENSOR.DEF;
TIMER_Valid_On(PT:=CONF_Tim_Valid_On);
STATE_ON			:=	TIMER_Valid_On.Q;
(*indicateur actionneur activé STATE_OFF*)
TIMER_Valid_Off.IN	:=	((NOT VAR_On AND NOT VAR_Lam AND NOT CONF_DI_Off AND (NOT IN_On OR NOT CONF_DI_On) AND (NOT IN_Lam OR NOT CONF_DI_Lam)) OR
						(IN_OFF AND CONF_DI_Off)) AND NOT DEF_SENSOR.DEF;
TIMER_Valid_Off(PT:=CONF_Tim_Valid_Off);
STATE_Off			:=	TIMER_Valid_Off.Q;
(*indicateur actionneur activé STATE_LAM*)
TIMER_Valid_Lam.IN	:=	((VAR_Lam  AND NOT CONF_DI_Lam AND (NOT IN_On OR NOT CONF_DI_On) AND (NOT IN_Off OR NOT CONF_DI_Off)) OR
						(IN_Lam AND CONF_DI_Lam));
TIMER_Valid_Lam(PT:=CONF_Tim_Valid_Lam);
STATE_Lam			:=	TIMER_Valid_Lam.Q;
(*indicateur STATE_NOK*)
STATE_Nok			:=	DEF_ON.DEF OR DEF_Off.DEF OR DEF_Sensor.DEF OR DEF_Lam.DEF OR DEF_Off_auto.DEF OR DEF_On_Imposs.DEF OR
						DEF_Off_Imposs.DEF;

(*défaut d'ouverture*)
DEF_On.Condition	:= 	VAR_On AND NOT STATE_On AND (CONF_DI_Off OR CONF_DI_On OR CONF_DI_Lam) AND NOT RESET;
DEF_On();
(*défaut de fermeture*)
DEF_Off.Condition	:= 	NOT VAR_on AND NOT VAR_Lam AND NOT STATE_Off AND (CONF_DI_Off OR CONF_DI_On OR CONF_DI_LAm) AND NOT RESET;
DEF_Off();
(*défaut de position laminage*)
DEF_Lam.Condition	:= 	VAR_Lam AND NOT STATE_Lam AND (CONF_DI_Off OR CONF_DI_On OR CONF_DI_Lam) AND NOT RESET;
DEF_Lam();
(*défaut capteur*)
DEF_Sensor.Condition	:= 	IN_On AND IN_Off AND CONF_DI_Off AND CONF_DI_On AND NOT RESET;
DEF_Sensor();


(* Reset des ordres *)
IF M_On AND RCP_M_On THEN
	M_On 	:= FALSE;
END_IF;
IF M_Off AND RCP_M_Off THEN
	M_Off		 := FALSE;
END_IF;
IF M_Lam AND RCP_M_Lam THEN
	M_Lam	 := FALSE;
END_IF;

END_FUNCTION_BLOCK

// ---- POUs/Composant/POMPES/BLOCK_PPM.TcPOU
FUNCTION_BLOCK BLOCK_PPM

(* Gestion d'une pompe turbo ADIXEN avec controleur OBCV4 sur réseau profibus*)
(* TYPE OBJET = POMPE TURBO*)

(****************historique des versions*****************************)

(* Version 1-0 - SP/JPC - VERSION INIITIALE - 6844 DP650 N35*)
(* Version 2-0 - HG - Adaptation pour journal des évènements externe - 24/06/2011*)

(*************************************************************************)

VAR_INPUT
	MANUAL:					BOOL;				(* ~ (OPC : 1 : available for OPC-clients) *)		(* Mode de pilotage manuel *)
	RESET:					BOOL;														(* Condition de réiinitialisation de la fonction *)
	WATER:					BOOL;				(* ~ (OPC : 1 : available for OPC-clients) *)		(*indication de refrodissement de la pompe ok*)

	DEF_Arret_Auto:				PRCDEF;		(*01 - défaut d'arrêt automatique de la pompe*)
	DEF_Marche_imposs:			PRCDEF;		(*02 - défaut de marche de la pompe turbo non autorisée*)
	DEF_Arret_imposs:				PRCDEF;		(*03 - défaut d'arrêt de la pompe turbo non autorisée*)
	DEF_On:						PRCDEF;		(*04 - défaut de marche de la pompe*)
	DEF_Off:						PRCDEF;		(*05 - défaut d'arrêt de la pompe*)

	CO_On:						BOOL;			(*demande de marche de la pompe en mode automatique généré par la fonction qui gère la pompe*)

	(*conditions d'autorisation*)
	EN_On_INT:					BOOL:= TRUE;	(*condition d'autorisation de marche et de standby de la pompe donnée par la fonction qui gère la pompe*)
	EN_Off_INT:					BOOL:= TRUE;	(*condition d'autorisation d'arrêt de la pompe donnée par la fonction qui gère la pompe*)
	EN_On_EXT:					BOOL:= TRUE;	(*condition d'autorisation de marche et de standby externe*)
	EN_Off_EXT:					BOOL:= TRUE;	(*condition d'autorisation d'arrêt de la pompe donnée par la fonction qui gère la pompe*)

	IN_On:						BOOL;	(* ~ (OPC : 1 : available for OPC-clients) *)		(*entrée TOR pompe en marche*)
	OUT_On:						BOOL;	(* ~ (OPC : 1 : available for OPC-clients) *)		(* Marche pompe *)
END_VAR

VAR_INPUT PERSISTENT
	CONF_Tim_Valid_On:			TIME:=T#0ms;	(*temporisation de validation du l'état STATE_OK*)
	CONF_Tim_Valid_Off:			TIME:=T#0ms;	(*temporisation de validation de l'état STATE_AR*)

	(*Entité*)
	IsComponent:		BOOL;			(*entité : composant*)
	IdXML:			STRING;			(*nom entité : identifiant pour recherche dans dico*)
	TagXML:			UINT;			(*nom entité : identifiant pour recherche dans dico*)
	IdParent:			STRING;			(*MNEMO de l'appelant*)
	MNEMO:			STRING;			(*MNEMO de l'entité*)
END_VAR

VAR_OUTPUT
	RQ_Cool:						BOOL;												(* Demande de refroidissement de la pompe turbo*)

	(*variable d'état d'autorisation*)
	AUTOR_On_IHM:				BOOL;			(* ~ (OPC : 1 : available for OPC-clients) *)	(*indique que la mise en marche de la pompe est autorisée en mode manuel depuis l'IHM*)
	AUTOR_Off_IHM:				BOOL;			(* ~ (OPC : 1 : available for OPC-clients) *)	(*indique que l'arrêt de la pompe est autorisée en mode manuel depuis l'IHM*)

	STATE_Ec:					BOOL;			(* ~ (OPC : 1 : available for OPC-clients) *)	(*indique que la pompe est en marche et n'a pas atteint sa vitesse*)
	STATE_On:					BOOL;			(* ~ (OPC : 1 : available for OPC-clients) *)	(*indique que la pompe est en marche et à atteint sa vitesse*)
	STATE_NOK:					BOOL;			(* ~ (OPC : 1 : available for OPC-clients) *)	(*indique la présence d'un défaut sur la pompe ou que l'ordre de marche a été refusé*)
	STATE_Off:					BOOL;			(* ~ (OPC : 1 : available for OPC-clients) *)	(*indique que la pompe est à l'arrêt*)
	STATE_Ihm:					USINT;			(* ~ (OPC : 1 : available for OPC-clients) *)	(*code d'état de la pompe*)
END_VAR

VAR
	TIMER_Valid_On:				TON;
	TIMER_Valid_Off:				TON;
	(* Variables pour les sorties profibus *)

	(* Variables demande en mode manuel*)
	M_On:						BOOL;					(* ~ (OPC : 1 : available for OPC-clients) *)	(* Ordre marche/arrêt de la  pompe en mode manuel *)
	RCP_M_On:					BOOL;														(* bit de reception de l'ordre de marche en mode manuel*)
	VAR_On:						BOOL;														(* variable intermédiaire de marche de la pompe*)

	VAR_CPT:						BLOCK_CPT_TEMPS;
END_VAR

VAR_EXTERNAL
	MANUAL_SAFETY_OFF:		BOOL;				(*desactive les sécurités en mode manuel*)
END_VAR

DEF_Arret_Auto.IdXml			:=	'3';
DEF_Arret_Auto.TagXml			:=	10;

DEF_Marche_imposs.IdXml			:=	'3';
DEF_Marche_imposs.TagXml		:=	5;

DEF_Arret_imposs.IdXml			:=	'3';
DEF_Arret_imposs.TagXml			:=	8;

DEF_On.IdXml					:=	'3';
DEF_On.TagXml					:=	1;

DEF_Off.IdXml					:=	'3';
DEF_Off.TagXml					:=	3;

(* Gestion des ordres en mode manuel *)
RCP_M_On 				:=	M_On;

(*gestion des bits d'autorisation en mode manuel*)
AUTOR_On_IHM			:=	NOT RESET AND ((EN_On_INT AND EN_On_EXT AND WATER) OR MANUAL_SAFETY_OFF)
							AND NOT VAR_On  AND MANUAL;
AUTOR_Off_IHM			:=	NOT RESET  AND VAR_On  AND MANUAL
							AND (( EN_Off_EXT AND EN_Off_INT) OR MANUAL_SAFETY_OFF);

(* AFFECTATION DES SORTIES LOGIQUES *)


(*défaut d'arrêt automatique de la pompe *)
DEF_Arret_Auto.CONDITION :=     (NOT WATER
								OR  NOT EN_On_INT
								OR NOT EN_On_EXT)
								AND  OUT_On AND NOT RESET;
DEF_arret_auto.DELAY:=T#0ms;
DEF_Arret_Auto();

(* Défaut de marche de la pompe primaire non autorisée en automatique*)
DEF_marche_imposs.CONDITION:=	NOT MANUAL AND CO_On AND (NOT EN_On_INT OR NOT EN_On_EXT)
								AND NOT MANUAL AND NOT RESET;
DEF_marche_imposs.DELAY := T#0ms;
DEF_marche_imposs();

(* Défaut d'arrêt de la pompe primaire non autorisée en automatique*)
DEF_arret_imposs.CONDITION	:=	NOT MANUAL AND NOT CO_On AND VAR_ON AND( NOT EN_Off_INT OR NOT EN_Off_EXT)
								AND NOT RESET;
DEF_arret_imposs.DELAY := T#0ms;
DEF_arret_imposs();

(* ARRET POMPE*)
IF 		(NOT CO_On AND NOT MANUAL AND EN_Off_INT AND EN_Off_EXT)
		OR ( RCP_M_On AND AUTOR_Off_IHM) OR RESET OR DEF_arret_auto.DEF
		THEN
			Var_On 				:= 	FALSE;
(*MARCHE POMPES*)
ELSIF	( CO_On AND NOT MANUAL AND EN_On_INT AND EN_On_EXT)
		 OR 	( RCP_M_On AND AUTOR_On_IHM) THEN
			Var_On 				:= 	TRUE;
END_IF;

(*SORTIE MARCHE POMPE*)
OUT_On			:= 	WATER AND VAR_On;

(*DEMANDE DE REFROIDISSEMENT DE LA POMPE*)
RQ_Cool			:=	VAR_On;

(* Défaut de marche de la pompe*)
DEF_ON.CONDITION := OUT_On AND NOT IN_On;
DEF_ON();

(* Défaut d'arrêt de la pompe*)
DEF_Off.CONDITION := NOT OUT_On AND IN_On;
DEF_Off();

(*affectation des bits d'état*)
(*indicateur pompe en marche STATE_ON*)
TIMER_Valid_On.IN	:=	OUT_On AND IN_On;
TIMER_Valid_On(PT:=CONF_Tim_Valid_On);
STATE_ON			:=	TIMER_Valid_On.Q;
(*indicateur pompe à l'arrêt STATE_OFF*)
TIMER_Valid_Off.IN	:=	NOT OUT_On AND NOT IN_On;
TIMER_Valid_Off(PT:=CONF_Tim_Valid_Off);
STATE_Off			:=	TIMER_Valid_Off.Q;
STATE_Ec			:=	VAR_On AND NOT IN_On;
STATE_NOK			:=	DEF_Arret_imposs.DEF OR DEF_Marche_imposs.DEF OR DEF_Arret_auto.DEF OR DEF_On.DEF OR DEF_Off.DEF;

IF NOT out_on THEN
	STATE_Ihm := 0;
ELSIF out_on AND NOT IN_On THEN
	STATE_ihm := 1;
ELSIF out_on AND in_on THEN
	STATE_ihm:=2;
END_IF;

(*Gestion compteur*)
VAR_CPT(I_On:= STATE_On);

(* Reset des ordres*)
IF M_On AND RCP_M_On THEN
	M_On		:= FALSE;
END_IF;

END_FUNCTION_BLOCK

// ---- POUs/Composant/POMPES/BLOCK_PCR_CTI_OB.TcPOU
FUNCTION_BLOCK BLOCK_PCR_CTI_OB

(* Gestion d'un objet pompe cryo CTI avec controleur ON-BOARD*)
(* TYPE OBJET = POMPE CRYO*)

(****************historique des versions************************************)

(* Version 1-0 - SP - 09/2010 -  VERSION INIITIALE - 6844 DP650 N35*)
(* Version 2-0 - HG - 04/2011 -  Ajout regen sur option - 7015 CT200 n°2*)
(* Version 3-0 - HG - 06/2011 - Adaptation pour journal des évènements externe*)
(* Version 3-1 - HG - 12/2012 - Modification défaut désamorçage pour cryo network (envoi OUT_On pendant regen)*)
(* Version 3-2 - GV - 07/2015 - Modification défaut arret auto (var_on modifié par Out_On)*)
(* Version 3-3 - LDS - 07/2015 - ajout d'un "forcage automatique" du CO_ETAT cryo*)
(********************************************************************************)

VAR_INPUT
	MANUAL:					BOOL;		(* Mode de pilotage manuel *)
	RESET:					BOOL;		(* Condition de réiinitialisation de la fonction *)
	WATER:					BOOL;		(*indication de refrodissement de la pompe ok*)

	DEF_Desamorcage:		PRCDEF;		(*01 - défaut désamorçage de la pompe cryogénique*)
	DEF_Arret_Auto:			PRCDEF;		(*02 - défaut d'arrêt automatique de la pompe*)
	DEF_Marche_imposs:		PRCDEF;		(*03 - défaut de marche de la pompe cryo non autorisée*)
	DEF_On:					PRCDEF;		(*04 - défaut de marche de la pompe*)
	DEF_Off:				PRCDEF;		(*05 - défaut d'arrêt de la pompe*)

	CO_On:					BOOL;		(*demande de marche de la pompe en mode automatique généré par la fonction qui gère la pompe*)
	CO_Regen:				BOOL;		(*demande de régénération de la pompe en mode automatique par la fonction qui gère la pompe*)

	IN_ST11:				BOOL;		(*indique que la pompe cryogénique est opérationnelle*)
	IN_ST12:				BOOL;		(*indique que la pompe cryogénique est en régénration*)
	IN_ON:					BOOL;		(*indique que la pompe cryogénique est en marche*)

	(*conditions d'autorisation*)
	EN_On_INT:					BOOL:= TRUE;	(*condition d'autorisation de marche de la pompe donnée par la fonction qui gère la pompe*)
	EN_Off_INT:					BOOL:= TRUE;	(*condition d'autorisation d'arrêt de la pompe donnée par la fonction qui gère la pompe*)
	EN_On_EXT:					BOOL:= TRUE;	(*condition d'autorisation de marche externe*)
	EN_Off_EXT:					BOOL:= TRUE;	(*condition d'autorisation d'arrêt de la pompe donnée par la fonction qui gère la pompe*)
	EN_Regen_INT:				BOOL:= TRUE;	(*condition d'autorisation de régénération de la pompe donnée par la fonction qui gère la pompe*)
	EN_Regen_EXT:				BOOL:= TRUE;	(*condition d'autorisation de régénération externe*)
	
	PRM_Forcage_Cryo_EXT:			BOOL;   
	PRM_Forcage_Cryo_INT:			BOOL;   	  		
END_VAR

VAR_INPUT PERSISTENT
	(*Entité*)
	IsComponent:		BOOL;			(*entité : composant*)
	IdXML:				STRING;			(*nom entité : identifiant pour recherche dans dico*)
	TagXML:				UINT;			(*nom entité : identifiant pour recherche dans dico*)
	IdParent:			STRING;			(*MNEMO de l'appelant*)
	MNEMO:				STRING;			(*MNEMO de l'entité*)
END_VAR

VAR_OUTPUT
	RQ_Cool:					BOOL;			(* Demande de refroidissement de la pompe cryogénique*)

	(*variable d'état d'autorisation*)
	AUTOR_On_IHM:				BOOL;			(*indique que la mise en marche de la pompe est autorisée en mode manuel depuis l'IHM*)
	AUTOR_Off_IHM:				BOOL;			(*indique que l'arrêt de la pompe est autorisée en mode manuel depuis l'IHM*)
	AUTOR_Regen_IHM:			BOOL;			(*indique que la régénération de la pompe est autorisée en mode manuel depuis l'IHM*)

	STATE_On:					BOOL;			(*indique que la pompe est en marche*)
	STATE_Ok:					BOOL;			(*indique que la pompe est en marche et à atteint sa température*)
	STATE_Nok:					BOOL;			(*indique la présence d'un défaut sur la pompe ou que l'ordre de marche a été refusé*)
	STATE_Ar:					BOOL;			(*indique que la pompe est à l'arrêt*)
	STATE_Ready:				BOOL;			(*indique que la pompe est prête à fonctionner*)
	STATE_Regen:				BOOL;			(*indique que la pompe est en régénération*)
	STATE_Ihm:					USINT;			(*code d'état de la pompe turbo*)
												(* 	0 = pompe à l'arrêt
												   	1 = pompe en régénération
													2 = amorcage en cours
													3 = pompe amorcée 
												*)
END_VAR

VAR

	(* Variables pour les sorties*)
	OUT_On:						BOOL;			(* Start pump *)
	OUT_Regen:					BOOL;			(* Regen pump *)

	(* Variables demande en mode manuel*)
	M_On:						BOOL;			(* Ordre marche pompe en mode manuel *)
	M_Regen:					BOOL;			(* Ordre regénération pompe en mode manuel *)

	RCP_M_On:					BOOL;			(*bit de reception de l'ordre de marche/arrêt en mode manuel*)
	RCP_M_Regen:				BOOL;			(*bit de reception de l'ordre de regeneration en mode manuel*)

	VAR_On:						BOOL;			(*bit intermédiaire de demande de marche de la pompe turbo*)
	VAR_Regen:					BOOL;			(*bit intermédiaire de demande de regeneration de la pompe turbo*)
	VAR_mem_ok:					BOOL;

	VAR_CPT:					BLOCK_CPT_TEMPS;
	
	Tempo_on_Cryo: 				TON;
END_VAR

VAR_EXTERNAL
	MANUAL_SAFETY_OFF:			BOOL;			(*desactive les sécurités en mode manuel*)
END_VAR

IdXML						:=	'1';
TagXML						:=	9;

DEF_Desamorcage.IdXml		:=	'16';
DEF_Desamorcage.TagXml		:=	12;

DEF_Arret_Auto.IdXml		:=	'3';
DEF_Arret_Auto.TagXml		:=	10;

DEF_Marche_imposs.IdXml		:=	'3';
DEF_Marche_imposs.TagXml	:=	5;

DEF_On.IdXml				:=	'3';
DEF_On.TagXml				:=	1;

DEF_Off.IdXml				:=	'3';
DEF_Off.TagXml				:=	3;


(* Gestion des ordres en mode manuel *)
	RCP_M_On 			:=	M_On;
	RCP_M_Regen			:=	M_Regen;

(*gestion des bits d'autorisation en mode manuel*)
	AUTOR_On_IHM			:=	NOT RESET AND NOT VAR_On  AND MANUAL
								AND ((EN_On_INT AND EN_On_EXT AND WATER) OR MANUAL_SAFETY_OFF);
	AUTOR_Off_IHM			:=	NOT RESET  AND VAR_On  AND MANUAL
								AND (( EN_Off_EXT AND EN_Off_INT) OR MANUAL_SAFETY_OFF);
	AUTOR_Regen_IHM			:=	NOT RESET  AND NOT VAR_Regen AND MANUAL (*AND VAR_On  *)
								AND (( EN_Regen_EXT AND EN_Regen_INT) OR MANUAL_SAFETY_OFF);

(*défaut d'arrêt automatique de la pompe*)
	DEF_Arret_Auto.CONDITION :=             (NOT WATER
									OR  NOT EN_On_INT
									OR NOT EN_On_EXT)
									AND OUT_On AND NOT RESET;
	DEF_arret_auto.DELAY:=T#0ms;
	DEF_Arret_Auto();

(* Défaut de marche de la pompe turbo non autorisée en automatique*)
	DEF_marche_imposs.CONDITION:=	NOT MANUAL AND CO_On AND( NOT EN_On_INT OR NOT EN_On_EXT)
									AND NOT MANUAL AND NOT RESET AND NOT VAR_On;
	DEF_marche_imposs.DELAY := T#0ms;
	DEF_marche_imposs();

(* ARRET POMPE*)
	IF 		(NOT CO_On AND NOT MANUAL AND EN_Off_INT AND EN_Off_EXT)
			OR ( RCP_M_On AND AUTOR_Off_ihm)
			OR RESET
			OR DEF_arret_auto.DEF
			THEN
					VAR_On 				:= 	FALSE;
					VAR_Regen			:=	FALSE;
(*MARCHE POMPES*)
	ELSIF	(CO_On AND NOT MANUAL AND EN_On_INT AND EN_On_EXT)
			 OR 	( RCP_M_On AND AUTOR_On_IHM) THEN
					VAR_On 				:= 	TRUE;
	END_IF
(*REGEN POMPES*)
	IF	( CO_Regen AND NOT MANUAL AND EN_Regen_INT AND EN_Regen_EXT)
			 OR 	( RCP_M_Regen AND AUTOR_Regen_IHM) THEN
					VAR_Regen 			:= 	TRUE;
	ELSIF	(VAR_Regen AND STATE_Regen) THEN
					VAR_Regen			:=	FALSE;
	END_IF;

Tempo_on_Cryo.PT:=T#8S;
Tempo_on_Cryo.IN := OUT_On AND NOT IN_On AND NOT DEF_On.DEF;
PRM_Forcage_Cryo_INT := Tempo_on_Cryo.Q;

(*SORTIE MARCHE POMPE*)
	OUT_On			:= 	WATER AND VAR_On AND NOT PRM_Forcage_Cryo_INT AND NOT PRM_Forcage_Cryo_EXT;
(*SORTIE REGEN POMPE*)
	OUT_Regen		:= 	VAR_Regen;
(*DEMANDE DE REFROIDISSEMENT DE LA POMPE*)
	RQ_Cool			:=	VAR_On;

(* Défaut désamorçage *)
		IF OUT_On AND IN_ST11 AND NOT IN_ST12 THEN
			VAR_Mem_Ok := TRUE;
		END_IF;
		IF NOT OUT_On OR VAR_Regen THEN
			VAR_Mem_Ok :=	FALSE;
		END_IF;

		DEF_Desamorcage.DELAY  := T#5s;
		DEF_Desamorcage.CONDITION := VAR_MEM_Ok AND NOT IN_ST11;
		DEF_Desamorcage();

(* Défaut de marche de la pompe*)
		DEF_ON.CONDITION := WATER AND VAR_On AND NOT IN_On;
		DEF_ON.DELAY:=T#15s;
		DEF_ON();

(* Défaut d'arrêt de la pompe*)
		DEF_OFF.CONDITION := NOT OUT_On AND IN_On AND NOT RESET;
		DEF_OFF.DELAY := T#10s;
		DEF_OFF();

(*affectation des bits d'état*)
	STATE_On			:=	OUT_On;
	STATE_Ok			:=	IN_ST11 AND OUT_On AND IN_On AND NOT IN_ST12;
	STATE_Regen			:=	IN_ST12;
	STATE_AR 			:= 	NOT OUT_On;
	STATE_NOK			:=	DEF_Desamorcage.DEF OR
							DEF_Marche_imposs.DEF OR
							DEF_Arret_auto.DEF OR
							DEF_On.DEF OR
							DEF_Off.DEF;
	STATE_Ready			:=	TRUE;

	IF STATE_Ar THEN
		STATE_Ihm	:=	0;
	ELSIF STATE_regen THEN
		STATE_Ihm 	:=	1;
	ELSIF STATE_on AND NOT STATE_ok THEN
		STATE_Ihm	:= 	2;
	ELSIF STATE_On AND STATE_Ok THEN
		STATE_ihm 	:= 	3;
	ELSE
		STATE_ihm 	:=	0;
	END_IF;


(*Gestion compteur*)
VAR_CPT(I_On:= STATE_On);

(* Reset des ordres *)
IF M_On AND RCP_M_On THEN
	M_On		 := FALSE;
END_IF;
IF M_Regen AND RCP_M_Regen THEN
	M_Regen	 := FALSE;
END_IF;

END_FUNCTION_BLOCK

// ---- POUs/Composant/VANNES/BLOCK_VVAT_650_NO.TcPOU
FUNCTION_BLOCK BLOCK_VVAT_650_NO

(* Gestion d'une vanne 3 positions VAT*)

(****************historique des versions*****************************)

(* Version 1-0 - SP - VERSION INITIALE*)
(* Version 1-1 - AB - VERSION INTERFACE STANDARD - 6970*)
(* Version 1-2 - JPC - OFFSET AUTO ADAPTATIF POUR REGULATION PRESSION *)
(* Version 2-0 - 05/2026 - MS - Adaptation pour journal des évènements externe*)

(*************************************************************************)


VAR_INPUT
(*paramètre standard*)
	RESET:   					BOOL; 											(*Condition RAZ actionneur*)
	MANUAL:  					BOOL; 	(* ~ (OPC : 1 : available for OPC-clients) *)		(*Mode manuel*)
	//MNEMO:						STRING;				(* ~ (OPC : 1 : available for OPC-clients) *)


(*entrée externe*)
	IN_OFF:						BOOL; 	(* ~ (OPC : 1 : available for OPC-clients) *)		(*E.TOR vanne fermée*)
	IN_ON:						BOOL; 	(* ~ (OPC : 1 : available for OPC-clients) *)		(*E.TOR vanne ouverte*)
	IN_POSITION:				ANALOG_INPUT;						 			(*E.Analogique retour position de la vanne*)
	I_PRESSION:					REAL;											(*Mesure de pression externe*)

(*Paramètres*)
	PRM_Mode:					BOOL; 	(* ~ (OPC : 1 : available for OPC-clients) *)		(*Mode FALSE = Position / TRUE = Pression*)
	PRM_Pression:				REAL; 	(* ~ (OPC : 1 : available for OPC-clients) *)		(*Consigne de pression - en unité cohérente avec la mesure*)
	PRM_Position:				REAL;	(* ~ (OPC : 1 : available for OPC-clients) *)		(*Consigne de position de la vanne en %*)
	PRM_W_Pr_HI:				REAL;	(* ~ (OPC : 1 : available for OPC-clients) *)		(*Tolérance haute de stabilisation de pression pour obtention de l'état stab pression ok*)
	PRM_W_Pr_LO:				REAL;	(* ~ (OPC : 1 : available for OPC-clients) *)		(*Tolérance basse de dtabilisation de pression pour obtention de l'état stab pression ok*)
	PRM_Tim_W_Pr:				TIME;	(* ~ (OPC : 1 : available for OPC-clients) *)		(*Temps de validation de stabilisation de la pression*)

(*défaut du bloc*)
	DEF_On:  					PRCDEF; 										(*00 - Défaut d'ouverture de la vanne*)
	DEF_Off:   					PRCDEF; 										(*01 - Défaut de fermeture de la vanne*)
	DEF_On_Imposs:				PRCDEF;										(*03 - Défaut d'ouverture ou de mise en laminage non autorisée en mode automatique*)
	DEF_Off_Imposs:				PRCDEF;										(*04 - Défaut de fermeture non autorisée en mode automatique*)
	DEF_Off_auto:				PRCDEF;										(*05 - Défaut de fermeture automatique de la vanne*)
	DEF_Position:				PRCDEF;										(*06 - Défaut d'obtention de la position*)
	DEF_Pression:				PRCDEF;										(*07 - Défaut d'obtention de la pression*)
	DEF_Surv_Pression:			PRCDEF;										(*08 - Défaut de surveillance de la pression - perte du critère de stabilisation*)
	ALA_Surv_Pression:			PRCDEF;										(*09 - Alarme de surveillance de la rpession - perte du critère de stabilisation*)

(*parametre de pilotage en entrée*)
	CO_On:   						BOOL; 											(*Ordre mode automatique ouverture*)
	CO_Lam:						BOOL;											(*Ordre mode automatique laminage*)
	EN_On_INT:   				BOOL;											(*Condition d'autorisation d'ouverture ou de laminage donnée par le bloc qui instancie le bloc actuator*)
	EN_Off_INT:  					BOOL; 											(*Condition d'autorisation de fermeture donnée par le bloc qui instacie le bloc actuator*)
	EN_On_EXT:					BOOL:=TRUE;									(*condition d'autorisation d'ouverture ou de laminage externe*)
	EN_Off_EXT:					BOOL:=TRUE;									(*condition d'autorisation de fermeture externe*)
END_VAR

VAR_INPUT PERSISTENT
(*parametre de configuration constructeur*)
(*les parametres suivants dépendent de la configuration de la machine*)
	CONF_Tim_Valid_On:  			TIME:=T#100ms; 			(*Temps validation de la position ouverte *)
	CONF_Tim_Valid_Off:   		TIME:=T#100ms; 			(*Temps validation de la position fermée *)
	CONF_EN_On:				USINT:=0;				(*définit la réaction du système en cas de perte des conditions d'autorisation d'activation EN_On*)
														(* 0 = désactivation automatique  en cas de perte des conditions d'autorisation d'activation uniquement en manuel*)
														(* 1 = désactivation automatique en cas de perte des conditions d'autorisation d'activation en auto et en manuel*)
														(* 2 = Pas de déscativation automatique*)
	CONF_Pr_Max_SP:			REAL;					(* Consigne max. de pression en pleine echelle 10V - correspond à la pleine échelle du capteur connecté au coffret*)
	CONF_WPos:				REAL;					(*Tolérance de positionnement pour obtention de l'état STATE_POS_ok*)
	CONF_Tim_WPos:			TIME;					(*Temps de validation de l'état STATE_POS_Ok*)
	PRM_Max_Tim_W:			TIME;	(* ~ (OPC : 1 : available for OPC-clients) *)		(*Temps Max d'obtention de l'état stabilisation pression ok*)
	PRM_Tim_Def_Pr:				TIME;	(* ~ (OPC : 1 : available for OPC-clients) *)		(*Temps d'enveloppe du défaut de surveillance de la pression*)
	PRM_Tim_Ala_Pr:				TIME;	(* ~ (OPC : 1 : available for OPC-clients) *)		(*Temps d'enveloppe de l'alarme de surveillance de la pression*)
	
	(*Entité*)
	IsComponent:				BOOL;		(*entité : composant*)
	IdXML:						STRING;		(*nom entité : identifiant pour recherche dans dico*)
	TagXML:						UINT;		(*nom entité : identifiant pour recherche dans dico*)
	IdParent:					STRING;		(*MNEMO de l'appelant*)
	MNEMO:						STRING;		(*MNEMO de l'entité*)

END_VAR

VAR_OUTPUT
	OUT_On: 					BOOL;	(* ~ (OPC : 1 : available for OPC-clients) *)		(*SORTIE Ouverture vanne*)
	OUT_Off:						BOOL; 	(* ~ (OPC : 1 : available for OPC-clients) *)		(*SORTIE Fermeture vanne*)
	OUT_Mode:					BOOL;	(* ~ (OPC : 1 : available for OPC-clients) *)		(*SORTIE sélection mode: FALSE = Position / TRUE = Pression *)
	OUT_SetPoint:				ANALOG_OUTPUT;								(*SORTIE ANA consigne position ou pression*)

	STATE_On:	   				BOOL; 	(* ~ (OPC : 1 : available for OPC-clients) *)		(*Indicateur ouverture ok*)
	STATE_Off:  					BOOL; 	(* ~ (OPC : 1 : available for OPC-clients) *)		(*Indicateur fermeture ok*)
	STATE_Nok:					BOOL;	(* ~ (OPC : 1 : available for OPC-clients) *)		(*Indicateur défaut sur la vanne*)
	STATE_Lam:					BOOL;	(* ~ (OPC : 1 : available for OPC-clients) *)		(*Indicateur mise en laminage ok *)
	STATE_Pos_Ok:				BOOL;	(* ~ (OPC : 1 : available for OPC-clients) *)		(*Indicateur de positionnement de la vanne ok *)
	STATE_Press_Ok:			BOOL;	(* ~ (OPC : 1 : available for OPC-clients) *)		(*Indicateur de stabilisation de la pression ok *)
	STATE_Ok:					BOOL;	(* ~ (OPC : 1 : available for OPC-clients) *)		(*Indicateur de stabilisation autour du point de consigne de pression
																				ou de positionnement ok si le controle est en mode position*)
	STATE_Position:				REAL;	(* ~ (OPC : 1 : available for OPC-clients) *)		(*Retour de position de la vanne*)
	STATE_Setpoint:				REAL;	(* ~ (OPC : 1 : available for OPC-clients) *)		(*Valeur de la consigne de pression ou position demandée*)
	STATE_Mode:				BOOL;	(* ~ (OPC : 1 : available for OPC-clients) *)		(*Mode de régulation en cours*)

	AUTOR_On_IHM:				BOOL; 	(* ~ (OPC : 1 : available for OPC-clients) *)		(*etat ouverture autorisée depuis la supervision en mode manuel*)
	AUTOR_Off_IHM:				BOOL; 	(* ~ (OPC : 1 : available for OPC-clients) *)		(*etat fermeture autorisée depuis la supervision en mode manuel*)
	AUTOR_Lam_IHM:			BOOL;	(* ~ (OPC : 1 : available for OPC-clients) *)		(*etat laminage autorisée depuis la supervision en mode manuel*)
	AUTOR_On_PLC:				BOOL;											(*etat ouverture autorisée depuis l'automate*)
	AUTOR_Off_PLC:				BOOL;											(*etat fermeture autorisée depuis l'automate*)
END_VAR


VAR
	TIMER_Valid_On:				TON;
	TIMER_Valid_Off:				TON;
	TIMER_Valid_Pos_ok:			TON;
	TIMER_Valid_Press_ok:		TON;

	M_On:  						BOOL; 	(* ~ (OPC : 1 : available for OPC-clients) *)		(*Ordre mode manuel ouverture de la vanne*)
	M_Off:   						BOOL; 	(* ~ (OPC : 1 : available for OPC-clients) *)		(*Ordre mode manuel fermeture de la vanne*)
	M_Lam:   					BOOL; 	(* ~ (OPC : 1 : available for OPC-clients) *)		(*Ordre mode manuel de mise en position laminage*)
	RCP_M_On:   					BOOL;
	RCP_M_Off:  					BOOL;
	RCP_M_Lam:					BOOL;
	VAR_On:						BOOL;											(*bit intermédiaire de demande d'ouverture de la vanne*)
	VAR_Lam:					BOOL;											(*bit intermédiaire de demande de mise en laminage de la vanne*)
	VAR_Mem_PRM_Pression:		REAL;											(*variable de mémorisation de la consigne de pression*)
	VAR_Prm_Pression_modifie:	BOOL;											(*variable activée à chaque changement de consigne de pression*)
	VAR_Attente_Stab:			BOOL;											(*variable activée aprés chaque demande de changement de consigne lorsque
																				la stabilisation de pression est attendue*)
	VAR_Surv_Pression:			BOOL;(*variable indiquant que la pression doit être surveillée - stabilisation atteinte*)

	VAR_OFFSET:				REAL;
	TEMPO_OFFSET:				TON;
	test:							BOOL;
END_VAR

VAR_EXTERNAL
	MANUAL_SAFETY_OFF:		BOOL;											(*desactive les sécurités en mode manuel*)
END_VAR


DEF_On.IdXml					:=	'3';
DEF_On.TagXml					:=	2;

DEF_Off.IdXml					:=	'3';
DEF_Off.TagXml					:=	4;

DEF_On_Imposs.IdXml				:=	'3';
DEF_On_Imposs.TagXml			:=	7;

DEF_Off_Imposs.IdXml				:=	'3';
DEF_Off_Imposs.TagXml			:=	9;

DEF_Off_auto.IdXml				:=	'3';
DEF_Off_auto.TagXml				:=	11;

DEF_Position.IdXml				:=	'1';
DEF_Position.TagXml				:=	9;

DEF_Pression.IdXml				:=	'1';
DEF_Pression.TagXml				:=	8;

DEF_Surv_Pression.IdXml			:=	'1';
DEF_Surv_Pression.TagXml		:=	11;

ALA_Surv_Pression.IdXml			:=	'1';
ALA_Surv_Pression.TagXml		:=	10;
ALA_Surv_Pression.Groupe		:=	1;

(*Affectation des constantes*)
IN_Position.CONF_Min 		:=	0.0;				(*position min retour vanne*)
IN_Position.CONF_Max	:=	100.0;			(*position max retour vanne*)
IN_Position();

IF VAR_OFFSET = 0.0 THEN
	VAR_OFFSET := 1.0;
END_IF

(*Mémorisation de la consigne et détection de changement de consigne*)

VAR_Prm_Pression_modifie :=  (PRM_Pression <> VAR_Mem_PRM_pression) AND VAR_Lam AND PRM_MODE AND NOT MANUAL AND NOT RESET;;
IF VAR_Lam AND PRM_mode THEN
	VAR_Mem_PRM_Pression	:= PRM_Pression;
ELSE
	VAR_Mem_PRM_Pression := 0.0;
END_IF;
(*positionnement du bit d'attente de la stabilisation de pression aprés modification de la consigne de pression*)
IF VAR_Prm_Pression_modifie AND NOT MANUAL AND NOT RESET  THEN
	VAR_Attente_Stab := TRUE;
END_IF;

(* Réception des ordres en mode manuel*)
	RCP_M_On 			:=	M_On;
	RCP_M_Off			:=	M_Off;
	RCP_M_Lam			:=	M_Lam;

(*Autorisation*)
	AUTOR_On_IHM		:= 	MANUAL AND ((EN_On_INT AND EN_On_EXT)
							OR MANUAL_SAFETY_OFF) AND NOT RESET AND NOT VAR_On;
	AUTOR_Off_IHM		:= 	MANUAL AND ((EN_Off_INT AND EN_Off_EXT)  OR
							MANUAL_SAFETY_OFF) AND NOT RESET AND  (VAR_On OR VAR_Lam);
	AUTOR_Lam_IHM	:=	MANUAL AND ((EN_On_INT AND EN_On_EXT)
							OR MANUAL_SAFETY_OFF) AND NOT RESET AND NOT VAR_Lam;
	AUTOR_On_PLC		:=	NOT MANUAL AND (EN_On_INT AND EN_On_EXT)
							AND NOT RESET;
	AUTOR_Off_PLC		:= 	NOT MANUAL AND (EN_Off_INT AND EN_Off_EXT)
							AND NOT RESET;
(*defaut ouverture ou laminage impossible en mode automatique*)
	DEF_On_Imposs.CONDITION:=	(CO_On OR CO_Lam) AND NOT AUTOR_On_PLC AND NOT MANUAL;
	DEF_On_Imposs.DELAY := T#0ms;
	DEF_On_Imposs();
(*Defaut fermeture impossible en mode automatique*)
	DEF_Off_Imposs.CONDITION:=	NOT CO_On AND NOT CO_Lam AND NOT AUTOR_Off_PLC AND NOT MANUAL
								AND (VAR_Lam OR VAR_On);
	DEF_Off_Imposs.DELAY := T#0ms;
	DEF_Off_Imposs();
(*defaut de fermeture automatique de la vanne*)
	DEF_Off_Auto.CONDITION :=             (NOT EN_On_INT OR NOT EN_On_EXT) AND  (VAR_On OR VAR_Lam)
								     AND ((CONF_En_ON=1) OR ((CONF_EN_On=0) AND MANUAL)) AND NOT RESET;
	DEF_Off_auto.DELAY:=T#0ms;
	DEF_Off_Auto();
(*gestion des sorties*)
IF 		(RCP_M_On AND AUTOR_On_IHM) OR
		(CO_On AND AUTOR_On_PLC) THEN
				VAR_On		:= 	TRUE;
				VAR_Lam	:= 	FALSE;
ELSIF 	(RCP_M_Lam AND AUTOR_Lam_IHM) OR
	    	(CO_Lam AND AUTOR_On_PLC) THEN
				VAR_On		:=	FALSE;
				VAR_LAm	:=	TRUE;
ELSIF 	RESET  OR DEF_Off_Auto.DEF OR
		(RCP_M_Off AND AUTOR_Off_IHM) OR
	    	((NOT CO_Lam AND NOT CO_On) AND AUTOR_Off_PLC) THEN
				VAR_On		:= 	FALSE;
				VAR_Lam	:=	FALSE;
END_IF;

OUT_On		:=	VAR_On;
OUT_Mode	:=	(VAR_Lam AND PRM_Mode);
OUT_Off		:=	VAR_Lam OR VAR_On;

(*Gestion de la consigne analogique pression ou position*)
IF 		PRM_Mode AND VAR_Lam THEN
			OUT_SetPoint.CONF_Max 	:= CONF_Pr_MAX_SP;
			OUT_SetPoint.CONF_Min	:= 0.0;

			IF NOT (I_PRESSION  <=  PRM_Pression * 1.03  AND I_PRESSION  >=  PRM_Pression *0.97) THEN
				TEMPO_OFFSET.PT	:=	T#1s;
				TEMPO_OFFSET.IN	:=	TRUE;
				IF TEMPO_OFFSET.Q THEN
					IF I_PRESSION  < PRM_Pression THEN
						VAR_OFFSET	:=	VAR_OFFSET + 0.01;
					ELSIF I_PRESSION  > PRM_Pression THEN
						VAR_OFFSET	:=	VAR_OFFSET - 0.01;
					ELSIF TRUE THEN
						VAR_OFFSET	:=	1.0;
					END_IF
					TEMPO_OFFSET.IN	:=	FALSE;
				END_IF
			ELSE
				TEMPO_OFFSET.IN	:=	FALSE;
			END_IF
			TEMPO_OFFSET();
			IF VAR_OFFSET > 2.0 OR VAR_OFFSET < 0.0 THEN
				VAR_OFFSET := 1.0;
			END_IF
			(*IF PRM_Pression < 0.1 AND PRM_Pression > 0.01 THEN
				OUT_SetPoint.Value		:= PRM_Pression*0.95;
			END_IF
			IF PRM_Pression < 0.01 AND PRM_Pression > 0.001 THEN
				OUT_SetPoint.Value		:= PRM_Pression*0.80;
			END_IF*)
			OUT_SetPoint.Value		:= PRM_Pression*VAR_OFFSET;
ELSIF 	NOT PRM_Mode AND VAR_Lam THEN
			OUT_SetPoint.CONF_Max 	:= 100.0;
			OUT_SetPoint.CONF_Min	:= 0.0;
			OUT_SetPoint.Value		:= PRM_Position;
ELSIF NOT VAR_Lam	THEN
			OUT_SetPoint.CONF_Max 	:= 100.0;
			OUT_SetPoint.CONF_Min	:= 0.0;
			OUT_SetPoint.Value		:= 0.0;
END_IF;
OUT_Setpoint();




(*indicateur actionneur activé STATE_ON*)
TIMER_Valid_On.IN	:=	VAR_ON AND IN_On;
TIMER_Valid_On(PT:=CONF_Tim_Valid_On);
STATE_ON			:=	TIMER_Valid_On.Q;
(*indicateur actionneur activé STATE_OFF*)
TIMER_Valid_Off.IN	:=	NOT VAR_Lam AND NOT VAR_On AND IN_off;
TIMER_Valid_Off(PT:=CONF_Tim_Valid_Off);
STATE_Off			:=	TIMER_Valid_Off.Q;
(*indicateur STATE_NOK*)
STATE_Nok			:=	DEF_ON.DEF OR DEF_Off.DEF OR DEF_Off_auto.DEF OR DEF_On_Imposs.DEF OR
						DEF_Off_Imposs.DEF OR DEF_pression.DEF OR DEF_Position.DEF;

(*temporisation de validation de la stabilisation à la consigne de position*)
TIMER_Valid_Pos_OK.IN		:=	VAR_Lam AND NOT PRM_Mode AND(  (ABS(IN_Position.Value - PRM_position) <= CONF_WPos) OR (CONF_WPos = 0.0));
TIMER_Valid_Pos_OK.PT		:=	CONF_Tim_WPos;
Timer_Valid_pos_OK();
STATE_Pos_OK				:= 	TIMER_Valid_Pos_OK.Q;


(*temporisation de validation de la stabilisation à la consigne de pression*)
TIMER_Valid_Press_OK.IN		:=	VAR_Lam AND PRM_Mode AND (((I_Pression >= PRM_W_Pr_LO) AND (I_Pression <= PRM_W_Pr_HI))
								OR (PRM_Tim_W_Pr = T#0ms))
								AND NOT VAR_Prm_Pression_modifie ;
TIMER_Valid_Press_OK.PT		:=	PRM_Tim_W_Pr;
TIMER_Valid_Press_OK();
STATE_Press_OK				:=	TIMER_Valid_Press_ok.Q;

(*indicateur actionneur activé STATE_LAM*)
STATE_Lam						:=	(VAR_Lam AND PRM_Mode) OR (VAR_LAM AND NOT PRM_Mode AND STATE_Pos_ok);



STATE_Position		:=	IN_position.Value;
STATE_Setpoint		:=	OUT_Setpoint.Value;
STATE_Mode		:=	OUT_Mode;
STATE_Ok  			:= 	STATE_Pos_Ok OR STATE_Press_Ok;

(*positionnement du bit de validation de la surveillance de la pression
si la stabilisation de pression est obtenue*)
IF (VAR_Lam AND PRM_MODE AND STATE_Press_ok) AND NOT MANUAL AND NOT RESET  THEN
	VAR_Surv_Pression :=	TRUE;
END_IF;
(*RAZ du bit d'attente de la stabilisation de pression lorsque l'état de stabilisation pression a été atteint ou
que le mode régulation de pression n'est plus demandé*)
IF (VAR_Attente_stab AND STATE_Press_ok) OR RESET OR NOT (VAR_Lam AND PRM_Mode)  THEN
	VAR_Attente_Stab := FALSE;
END_IF;

(*RAZ du bit de surveillance de la stabilisation si pas en mode régulation de pression ou si un changement de consigne est apparu*)
IF VAR_Prm_Pression_modifie  OR RESET OR NOT (VAR_Lam AND PRM_Mode)  THEN
	VAR_Surv_Pression := FALSE;
END_IF;

(*défaut d'ouverture*)
	DEF_On.Condition			:= 	VAR_On AND NOT STATE_On;
	DEF_On();
(*défaut de fermeture*)
	DEF_Off.Condition			:= 	NOT VAR_on AND NOT VAR_Lam AND NOT STATE_Off;
	DEF_Off();
(*défaut d'obtention de la position*)
	DEF_Position.Condition	:= 	VAR_Lam AND NOT PRM_Mode AND NOT STATE_Pos_Ok;
	DEF_position();
(*défaut d'obtention de la pression - le défaut n'est plus surveillé lorsque l'état STATE_Press_ok a été atteint  et est
surveillé de nouveau aprés un changement de consigne*)
	DEF_Pression.Condition	:= 	VAR_Lam AND PRM_Mode AND NOT STATE_Press_Ok AND VAR_Attente_Stab
								AND NOT MANUAL AND NOT RESET;
	DEF_Pression(DELAY		:=	PRM_Max_Tim_W);

(*défaut de surveillance de la pression - l'état STATE_Press_Ok est perdu pendant un temps supérieur à PRM_TIM_SURV_PR *)
DEF_Surv_Pression.CONDITION	:=	VAR_Lam AND PRM_Mode AND NOT State_Press_OK AND VAR_Surv_Pression
								AND NOT MANUAL AND NOT RESET;
DEF_Surv_Pression (DELAY:=PRM_Tim_Def_Pr);


(*défaut de surveillance de la pression - l'état STATE_Press_Ok est perdu pendant un temps supérieur à PRM_ALA_SURV_PR*)
ALA_Surv_Pression.CONDITION 	:=	VAR_Lam AND PRM_Mode AND NOT State_Press_OK AND VAR_Surv_Pression
									AND NOT MANUAL AND NOT RESET;
ALA_Surv_Pression (DELAY:=PRM_Tim_Ala_Pr);
(* Reset des ordres *)
	IF M_On AND RCP_M_On THEN
		M_On 	:= FALSE;
	END_IF;
	IF M_Off AND RCP_M_Off THEN
		M_Off		 := FALSE;
	END_IF;
	IF M_Lam AND RCP_M_Lam THEN
		M_Lam		 := FALSE;
	END_IF;

END_FUNCTION_BLOCK

// ---- POUs/Composant/JAUGES/BLOCK_BCG450_ETHERCAT.TcPOU
FUNCTION_BLOCK BLOCK_BCG450_ETHERCAT


(* Gestion d'une jauge triple BCG450 INFICON avec interface ethercat*)

(****************historique des versions*****************************)

(* Version 1-0 - AB - version initiale développée sur 8760 CT100 n102 *)
(* Versoin basée sur BLOCK_BCG_450_ANA version 4-0 *)

(*************************************************************************)

VAR_INPUT
	I_PARAM_SYSTEM_OK:	BOOL;													(*paramétrage système ok*)
(*paramètre standard*)
	RESET:   				BOOL; 													(*Condition RAZ actionneur*)
	MANUAL:  				BOOL; 													(*Mode manuel*)

	IN_Pression: 				REAL; 					(* Retour pression *)
	IN_WcState	 AT%I*:		BOOL;					(*0 = Data valid, 1 = Data invalid*)

(*___________________TEST ETHERCAT___________________________*)
(*ACTIVE SENSOR NUMBER*)
	IN_Active_Sensor			AT%I*:	UINT;
(*READING VALID VALUE*)
	IN_Reading_Valid_M1		AT%I*:	BOOL;
	IN_Reading_Valid_M2		AT%I*:	BOOL;
	IN_Reading_Valid_M3		AT%I*:	BOOL;
	IN_Reading_Valid_M4		AT%I*:	BOOL;
(*SPECIFIC M4*)
	IN_Emission_State_M4		AT%I*:	BOOL;
	IN_Degas_State_M4		AT%I*:	BOOL;
(*WARNING/ALARM STATE*)
	IN_Overrange_M1 		AT%I*:	BOOL;
	IN_Underrange_M1 		AT%I*:	BOOL;
	IN_Overrange_M2 		AT%I*:	BOOL;
	IN_Underrange_M2 		AT%I*:	BOOL;
	IN_Overrange_M3 		AT%I*:	BOOL;
	IN_Underrange_M3 		AT%I*:	BOOL;
	IN_Overrange_M4 		AT%I*:	BOOL;
	IN_Underrange_M4 		AT%I*:	BOOL;
	IN_Active_Ex_Status		AT%I*:	USINT;
	IN_Active_Dev_War_Det	AT%I*:	UDINT;
	IN_Active_Man_War_Det	AT%I*:	UDINT;
	IN_Latched_Ex_Status		AT%I*:	USINT;
	IN_Latched_Man_War_Det	AT%I*:	UDINT;
	IN_Latched_Man_Err_Det	AT%I*:	UDINT;
(*______________________________________________________________*)

	CO_Stop:				BOOL;					(* Condition de forcage d'arrêt d'alimentation de la jauge *)
	CO_inhibe_Seuil:			BOOL;					(*information externe d'inhibition des seuils*)


	I_Stop_Rah:				BOOL;					(* information externe de demande d'arrêt de la mesure avant remise à la PAtm *)
	I_VHxx:					BOOL;					(* état des vannes de ventilation VH11 ou VH12 pour redémarrage temporisé de la mesure*)

	PRM_Tim_Stop:			TIME:=T#10s;				(*Temps de validation de l'arrêt de la jauge*)
	PRM_Tim_Restart:		TIME:=T#10s;				(*Temps pour remise en marche de la jauge
																							aprés reception de la condition I_Restart_Mesure*)
	PRM_Seuil: 				ARRAY[0..15] OF REAL;	(* Valeur des seuils*)
	PRM_Delais:				ARRAY[0..15] OF TIME;	(*Delais de validation du seuil en multiple de 100ms *)
	PRM_Type_seuil: 			ARRAY[0..15] OF BOOL; 	(* Type du seuil n°1 (False=seuil vide, True=seuil pression) *)


(*entrées d'autorisation*)
	EN_Dgz_EXT:			BOOL;			(*condition d'autorisation d'activation de la sortie de dégazage de la jauge externe*)
	EN_Off_EXT:				BOOL;			(*condition d'autorisation d'arrêt de la jauge externe*)

(*Défaut*)
	DEF_jauge:					PRCDEF;	(* indicateur de défaut de fonctionnement de la jauge  *)
	DEF_Pilotage:				PRCDEF;


END_VAR

VAR_OUTPUT
(*Variable d'état*)
	STATE_Seuil:		 		ARRAY[0..15] OF BOOL; 	(*Tableau des seuils*)
	STATE_Pression:				REAL; 		(* Valeur de la pression (dans l'unité sélectionnée) *)
	STATE_Ok:					BOOL;		(* Jauge à l'état OK*)
	STATE_Nok:					BOOL;		(* Jauge en défaut*)
	STATE_Err:					USINT;		(*Code d'erreur
																				0 = Pas d'erreur
																				1 = EEPROM Error Ou défaut jauge capacitive 
																				2 = Défaut jauge à cathode chaude
																				3 = Défaut jauge pirani *)


	O_Pret_Pour_Rah:				BOOL;											(*information d'arrêt avant rah de la mesure effectué - délivrée aprés arret
																				et une tempo égale à PRM_Tim_Stop ou si la pression est supérieure à 2e-2 mbar*)

(*Variable d'information d'autorisation*)
	AUTOR_Off_IHM:				BOOL;	(* ~ (OPC : 1 : available for OPC-clients) *)		(*Autorisation d'arrêt de la jauge depuis l'IHM en mode manuel*)
	AUTOR_On_IHM:				BOOL;	(* ~ (OPC : 1 : available for OPC-clients) *)		(*Autorisation de marche de la jauge depuis l'IHM en mode manuel*)
	AUTOR_Dgz_IHM:			BOOL;	(* ~ (OPC : 1 : available for OPC-clients) *)		(*Autorisation de dégazage depuis l'IHM en mode manuel*)
END_VAR

VAR
	OP_DGZ:					BLOCK_G7;		(* séquence de mise en dégazage de la jauge*)
	OP_RaH:					BLOCK_G7;		(* séquence d'arrêt filament pour remise à H de l'enceinte*)

	M_M1:						BOOL;	(* ~ (OPC : 1 : available for OPC-clients) *)		(*Ordre de marche / arret de la jauge en mode manuel*)
	M_DGZ:						BOOL;	(* ~ (OPC : 1 : available for OPC-clients) *)		(*Ordre de dégazage de la jauge en mode manuel*)
	RCP_M_M1:					BOOL;
	RCP_M_DGZ:				BOOL;

	VAR_Degas_Ok:				BOOL;			(*variable permettant de mémoriser que le dégazage a été effectué et remise à 0*)
(*
	VAR_Stop:					BOOL;			(*Variable intermediaire de gestion de la marche arrêt de la jauge en mode manuel*)

	VAR_Stop_Mesure:			BOOL;			(*Bit indiquant que la mesure est stoppée temporairement sur demande externe*)
	VAR_Dem_Dgz:				BOOL;			(*Bit de demande de dégazage en mode manuel*)
	VAR_Mem_Stop_Mesure:		BOOL;
*)

	i:							USINT;

	TIMER_Stop_Jauge:			TON;
	(*TIMER_Restart_Jauge:		TP;*)
	TIMER_Restart_Jauge:		TON;
	TIMER_Degas:				TON;
	TIMER_Seuil:					ARRAY[0..15] OF TON;
	Timer_Reprise_Pompage:		TON;

	TIMER_State_Ok:				TON;

	Timer_Envoi_CoE:			TON;
	WRITE_CoE_WORD:			WRITE_CoE_WORD;	(*fonction d'écriture de paramètres CoEde type word*)
	WRITE_CoE_BOOL:			WRITE_CoE_BOOL;	(*fonction d'écriture de paramètres CoE de type booléen*)

(*___________________TEST ETHERCAT___________________________*)
	VAR_Mem_Active_Ex:			BOOL;
	VAR_Mem_Active_Dev_War:	BOOL;
	VAR_Mem_Active_Man_War:	BOOL;
	VAR_Mem_Latched_Ex:		BOOL;
	VAR_Mem_Latched_Man_War:	BOOL;
	VAR_Mem_Latched_Man_Err:	BOOL;
(*______________________________________________________________*)
END_VAR


VAR_INPUT PERSISTENT
	CONF_Unit: 				USINT; 					(* Unité : 0=mb,1=mTorr,2=Pa *)
	CONF_degas_auto:		BOOL;					(* Option de degazage apres remise à atmosphere *)
	CONF_Tim_Degas:		TIME;					(* Durée d'activation de la sortie de dégazage*)

	(*variables CoE*)
	CONF_NetId:				T_AmsNetId;				(*on le trouve dans le .tsm, sur le device ethercat , onglet ethercat, champ NetId*)
	CONF_SlaveAddr:			UINT;					(*on le trouve dans le .tsm, sur le device jauge, onglet ethercat, champ Ethercat Addr*)


	(*Entité*)
	IsComponent:		BOOL;			(*entité : composant*)
	IdXML:			STRING;			(*nom entité : identifiant pour recherche dans dico*)
	TagXML:			UINT;			(*nom entité : identifiant pour recherche dans dico*)
	IdParent:			STRING;			(*MNEMO de l'appelant*)
	MNEMO:			STRING;			(*MNEMO de l'entité*)
END_VAR

IdXML					:=	'2';
TagXML					:=	2;

DEF_jauge.IdXml			:=	'1';
DEF_jauge.TagXml		:=	7;

DEF_Pilotage.IdXML		:=	'1';
DEF_Pilotage.TagXML		:=	25;


(*Reception des ordres de maintenance*)
RCP_M_M1		:= 	M_M1;
RCP_M_DGZ		:=	M_DGZ;

(*calcul pression *)
IF STATE_Ok THEN
	STATE_Pression := IN_Pression;
ELSE
	STATE_Pression := 0;
END_IF

(* états jauge *)
(*On temporise le state_ok car en cours de descente en vide lros du basculement dur cathode chaude on peut avoir un petit 0mbar transitoire*)
TIMER_State_Ok.PT	:=	T#3s;
(*signal correct ou RaH en cours (coupure filament en vide secondaire)*)
IF IN_Pression > 1.0E-12 OR OP_RAH.EC THEN
	TIMER_State_Ok.IN	:=	FALSE;
ELSE
	TIMER_State_Ok.IN	:=	TRUE;
END_IF
TIMER_State_Ok();


STATE_Ok	:= NOT TIMER_State_Ok.Q AND NOT IN_WcState;
STATE_Nok	:= DEF_jauge.DEF;


(* GESTION DES SEUILS *)
FOR i:=1 TO 15 DO
		TIMER_Seuil[i].PT		:=	PRM_Delais[i];
		TIMER_Seuil[i].IN		:=	(((STATE_Pression >= PRM_Seuil[i]) AND PRM_Type_seuil[i]) OR		(*Seuil en pression*)
								((STATE_Pression <= PRM_Seuil[i]) AND NOT PRM_Type_seuil[i]))		(*Seuil de vide*)
								AND NOT RESET AND NOT CO_inhibe_Seuil AND STATE_Ok;
		TIMER_Seuil[i]();
		STATE_Seuil[i]		:= 	TIMER_Seuil[i].Q;
END_FOR;

(* ---------------------------- gestion dégazage -------------------------------------*)
(* dégazage autorisé en mode manuel si le dégazage est autorisé et la pression inférieure à 6e-6 mbar et si la sortie n'est pas déjà active
et si mode manuel*)
AUTOR_Dgz_IHM		:=	MANUAL
						AND NOT RESET
						AND NOT OP_DGZ.EC
						AND ( STATE_Pression < 5E-6)
						AND EN_Dgz_EXT
						AND State_OK;

(* temporisation de dégazage*)
TIMER_Degas.PT	:= CONF_Tim_Degas;
TIMER_Degas.IN	:= OP_DGZ.Etape.3;
TIMER_Degas();

(*gestion du drapeau dégazage ok*)
IF OP_DGZ.Etape.0 THEN
	VAR_Degas_Ok := FALSE;
ELSIF OP_DGZ.OK THEN
	VAR_Degas_Ok := TRUE;
END_IF



(* ---------------------------- gestion marche / arrêt filament -------------------------------------*)
(*On interdit le pilotage en mode manuel (la mise en manu du filament n'est pas gérable ainsi, et en auto le filament va se rallumer tout seul)*)
AUTOR_Off_IHM := FALSE;
AUTOR_On_IHM := FALSE;

(*temporisation d'arrêt de la jauge*)
TIMER_Stop_Jauge.PT	:=	PRM_Tim_Stop;
TIMER_Stop_Jauge.IN	:=	OP_RaH.Etape.5;
TIMER_Stop_Jauge();

(*temporisation de redémarrage de la jauge ==> remise en auto du filament*)
(*Remarque : on n'allume pas le filament, donc tempo peut être courte, on squizze le PRM_tim_restart (mais reste dans l'interface standard pour anciens PRG_Pompage)*)
TIMER_Restart_Jauge.PT	:=	PRM_Tim_Restart;
TIMER_Restart_Jauge.IN	:=	OP_RaH.Etape.7;
TIMER_Restart_Jauge();

(*temporisation d'attente max d'ouverture de VH avant passage direct dans étape de remise en auto du filament
==> permet de contrer une reprise de pompage en cours de ventilation alors qu'on a déjà mis en off le filament*)
Timer_Reprise_Pompage.PT	:=	T#10s;
Timer_Reprise_Pompage.IN	:=	OP_RaH.Etape.6;
Timer_Reprise_Pompage();

(*interfaçage avec autres fonctions*)
O_Pret_Pour_Rah	:=	OP_RaH.Etape.6 OR (STATE_Pression > 0.02);


(* ---------------------------- gestion de l'envoi de données CoE -------------------------------------*)
(*Configuration de la fonction avec données inchangeantes*)
WRITE_CoE_WORD.IN_NetId			:=	CONF_NetId;
WRITE_CoE_WORD.IN_SlaveAddr		:=	CONF_SlaveAddr;
WRITE_CoE_BOOL.IN_NetId			:=	CONF_NetId;
WRITE_CoE_BOOL.IN_SlaveAddr		:=	CONF_SlaveAddr;

(*Remplissage  de données à envoyer selon étapes des G7*)
(*marche dégazage*)
IF OP_DGZ.Etape.1 THEN
	WRITE_CoE_WORD.IN_Index		:=	16#FB43;
	WRITE_CoE_WORD.IN_SubIndex	:=	01;
	WRITE_CoE_WORD.IN_Value		:=	16#0401;			(*la jauge prend 01 04 mais codage MSB ici*)

(*arrêt dégazage*)
ELSIF OP_DGZ.Etape.4 THEN
	WRITE_CoE_WORD.IN_Index		:=	16#FB43;
	WRITE_CoE_WORD.IN_SubIndex	:=	01;
	WRITE_CoE_WORD.IN_Value		:=	16#0400;			(*la jauge prend 00 04 mais codage MSB ici*)

(*arrêt du filament*)
ELSIF OP_RaH.Etape.3 THEN
	WRITE_CoE_WORD.IN_Index		:=	16#FB44;
	WRITE_CoE_WORD.IN_SubIndex	:=	01;
	WRITE_CoE_WORD.IN_Value		:=	16#0400;
END_IF


(*mise en manuel du filament*)
IF OP_RaH.Etape.1 THEN
	WRITE_CoE_BOOL.IN_Index		:=	16#8035;
	WRITE_CoE_BOOL.IN_SubIndex	:=	02;
	WRITE_CoE_BOOL.IN_Value		:=	16#1;

(*mise en automatique du filament*)
ELSIF OP_RaH.Etape.8 THEN
	WRITE_CoE_BOOL.IN_Index		:=	16#8035;
	WRITE_CoE_BOOL.IN_SubIndex	:=	02;
	WRITE_CoE_BOOL.IN_Value		:=	16#0;
END_IF

(*marche de la fonction*)
WRITE_COE_WORD.IN_ON		:=	OP_DGZ.Etape.1
								OR OP_DGZ.Etape.4
								OR OP_RaH.Etape.3;
WRITE_CoE_BOOL.IN_ON		:=	OP_RaH.Etape.1
								OR OP_RaH.Etape.8;

(*appel fonction*)
WRITE_CoE_WORD();
WRITE_CoE_BOOL();


(*parcours des G7*)
ACT_DGZ();
ACT_RAH();


(*Gestion défaut jauge*)
DEF_jauge.DELAY		:= T#5s;
DEF_jauge.CONDITION	:= NOT STATE_Ok AND NOT RESET;
DEF_jauge();

(* Gestion défaut pilotage jauge*)
DEF_Pilotage.DELAY		:=	T#0ms;
DEF_Pilotage.CONDITION	:=	OP_RaH.Etape.12 OR OP_DGZ.Etape.10;
DEF_Pilotage();



(*RAZ des ordres de maintenance*)
IF RCP_M_M1 AND M_M1 THEN
	M_M1:=FALSE;
END_IF;
IF RCP_M_Dgz AND M_Dgz THEN
	M_Dgz:=FALSE;
END_IF;

(*___________________TEST ETHERCAT___________________________*)
	IF IN_Active_Ex_Status > 0 THEN
		VAR_Mem_Active_Ex			:=	TRUE;
	END_IF
	IF IN_Active_Dev_War_Det > 0 THEN
		VAR_Mem_Active_Dev_War	:=	TRUE;
	END_IF
	IF IN_Active_Man_War_Det > 0 THEN
		VAR_Mem_Active_Man_War	:=	TRUE;
	END_IF
	IF IN_Latched_Ex_Status > 0 THEN
		VAR_Mem_Latched_Ex		:=	TRUE;
	END_IF
	IF IN_Latched_Man_War_Det > 0 THEN
		VAR_Mem_Latched_Man_War	:=	TRUE;
	END_IF
	IF IN_Latched_Man_Err_Det > 0 THEN
		VAR_Mem_Latched_Man_Err	:=	TRUE;
	END_IF
(*______________________________________________________________*)

ACTION ACT_DGZ:
OP_DGZ(
	N_STEP_OP_OK:= 6,
	N_STEP_OP_NOK:= 0);

(*GRAFCET*)
(* initialisation du grafcet*)
IF 		OP_DGZ.ETAPE = 0
		THEN
				OP_DGZ.ETAPE.0 := TRUE;
(*repositionnement sur étape 0 : reset ou pression supérieure à 100mbar mise à 0 du flag dgz ok)*)
ELSIF	(RESET OR STATE_Pression > 100)
		THEN
				OP_DGZ.ETAPE := 0;			(*RAZ grafcet*)
				OP_DGZ.ETAPE.0:=TRUE;
(*étape 0-1 : demande manuelle ou gestion automatique (si option) avec pression < 5e-6 mbar, jauge ok et autorisation externe*)
ELSIF 	OP_DGZ.ETAPE.0
		AND( (MANUAL AND RCP_M_DGZ)
			OR (NOT MANUAL AND (STATE_Pression < 5E-6) AND STATE_Ok AND EN_Dgz_EXT AND CONF_degas_auto)
			)
		THEN
				OP_DGZ.ETAPE.1:=TRUE;
				OP_DGZ.ETAPE.0:=FALSE;

(*étape 1-2 ==> envoi de la commande de mise en dgz réussie (au niveau de twincat)*)
ELSIF	OP_DGZ.Etape.1
		AND NOT WRITE_CoE_WORD.STATE_Busy
		AND NOT WRITE_CoE_WORD.STATE_Error
		THEN
				OP_DGZ.ETAPE.2:=TRUE;
				OP_DGZ.ETAPE.1:=FALSE;

(*étape 1-10 ==> envoi de la commande de mise en dgz échouée, on va en étape défaut *)
ELSIF	OP_DGZ.Etape.1
		AND NOT WRITE_CoE_WORD.STATE_Busy
		AND WRITE_CoE_WORD.STATE_Error
		THEN
				OP_DGZ.ETAPE.10:=TRUE;
				OP_DGZ.ETAPE.1:=FALSE;

(*étape 2-3 ==> libre *)
ELSIF	OP_DGZ.Etape.2
		THEN
				OP_DGZ.ETAPE.3:=TRUE;
				OP_DGZ.ETAPE.2:=FALSE;

(*étape 3-4 ==> attente temporisatrion de dégazage *)
ELSIF	OP_DGZ.Etape.3
		AND TIMER_Degas.Q
		THEN
				OP_DGZ.ETAPE.4:=TRUE;
				OP_DGZ.ETAPE.3:=FALSE;

(*étape 4-5 ==> envoi de la commande de arret dgz réussie (au niveau de twincat)*)
ELSIF	OP_DGZ.Etape.4
		AND NOT WRITE_CoE_WORD.STATE_Busy
		AND NOT WRITE_CoE_WORD.STATE_Error
		THEN
				OP_DGZ.ETAPE.5:=TRUE;
				OP_DGZ.ETAPE.4:=FALSE;

(*étape 4-10 ==> envoi de la commande de mise en dgz échouée, on va en étape défaut *)
ELSIF	OP_DGZ.Etape.4
		AND NOT WRITE_CoE_WORD.STATE_Busy
		AND WRITE_CoE_WORD.STATE_Error
		THEN
				OP_DGZ.ETAPE.10:=TRUE;
				OP_DGZ.ETAPE.4:=FALSE;

(*étape 5-6 ==> libre *)
ELSIF	OP_DGZ.Etape.5
		THEN
				OP_DGZ.ETAPE.6:=TRUE;
				OP_DGZ.ETAPE.5:=FALSE;

(*étape 6-1 ==> nouvel ordre de degazage manuel , en auto on ne relance pas, on fait aussi retomber le flag *)
ELSIF	OP_DGZ.Etape.6
		AND (MANUAL AND RCP_M_DGZ)
		THEN
				OP_DGZ.ETAPE.1:=TRUE;
				OP_DGZ.ETAPE.6:=FALSE;
				VAR_Degas_Ok := FALSE;

(*étape 10- 0 ==> pb envoi de la commande*)
ELSIF	OP_DGZ.Etape.10
		THEN
				OP_DGZ.Etape.0 := TRUE;
				OP_DGZ.Etape.10 := FALSE;

END_IF

OP_DGZ.POST();
END_ACTION

ACTION ACT_RAH:
OP_RAH(
	N_STEP_OP_OK:= 0,
	N_STEP_OP_NOK:= 0);

(*GRAFCET*)
(* initialisation du grafcet*)
IF 		OP_RaH.ETAPE = 0
		THEN
				OP_RaH.ETAPE.0 := TRUE;
(*repositionnement sur étape 0 : reset *)
ELSIF	RESET
		THEN
				OP_RAH.ETAPE := 0;			(*RAZ grafcet*)
				OP_RAH.ETAPE.0:=TRUE;
(*étape 0-1 : demande manuelle ou gestion automatique (si option) avec pression < 6.6e-2 mbar, jauge ok et autorisation externe*)
ELSIF 	OP_RAH.ETAPE.0
		AND I_Stop_Rah
		AND STATE_Pression < 0.02
		THEN
				OP_RAH.ETAPE.1:=TRUE;
				OP_RAH.ETAPE.0:=FALSE;

(*étape 1-2 ==> envoi de la commande de mise en mode manuel du pilotage filament (au niveau de twincat)*)
ELSIF	OP_RAH.Etape.1
		AND NOT WRITE_CoE_BOOL.STATE_Busy
		AND NOT WRITE_CoE_BOOL.STATE_Error
		THEN
				OP_RAH.ETAPE.2:=TRUE;
				OP_RAH.ETAPE.1:=FALSE;

(*étape 1-12 ==> envoi de la commande de mise en manuel échouée, on va en étape défaut *)
ELSIF	OP_RAH.Etape.1
		AND NOT WRITE_CoE_BOOL.STATE_Busy
		AND WRITE_CoE_BOOL.STATE_Error
		THEN
				OP_RAH.ETAPE.12:=TRUE;
				OP_RAH.ETAPE.1:=FALSE;

(*étape 2-3 ==> libre *)
ELSIF	OP_RAH.Etape.2
		THEN
				OP_RAH.ETAPE.3:=TRUE;
				OP_RAH.ETAPE.2:=FALSE;

(*étape 3-4 ==> envoi de la commande d'arrêt filament réussie *)
ELSIF	OP_RAH.Etape.3
		AND NOT WRITE_CoE_WORD.STATE_Busy
		AND NOT WRITE_CoE_WORD.STATE_Error
		THEN
				OP_RAH.ETAPE.4:=TRUE;
				OP_RAH.ETAPE.3:=FALSE;

(*étape 3-4 ==> envoi de la commande d'arrêt filament échouée *)
ELSIF	OP_RAH.Etape.3
		AND NOT WRITE_CoE_WORD.STATE_Busy
		AND WRITE_CoE_WORD.STATE_Error
		THEN
				OP_RAH.ETAPE.12:=TRUE;
				OP_RAH.ETAPE.3:=FALSE;

(*étape 4-5 ==> libre *)
ELSIF	OP_RAH.Etape.4
		THEN
				OP_RAH.ETAPE.5:=TRUE;
				OP_RAH.ETAPE.4:=FALSE;

(*étape 5-6 ==> temporisation d'arrêt jauge *)
ELSIF	OP_RAH.Etape.5
		AND TIMER_Stop_Jauge.Q
		THEN
				OP_RAH.ETAPE.6:=TRUE;
				OP_RAH.ETAPE.5:=FALSE;

(*étape 6-7 ==> après envoi de l'information O_Pret_RaH, on attend retour VH ouverte ou P>= 0.02*)
ELSIF	OP_RAH.Etape.6
		AND (I_VHxx OR (STATE_Pression >= 0.02))
		THEN
				OP_RAH.ETAPE.7:=TRUE;
				OP_RAH.ETAPE.6:=FALSE;

(*etape 6-8 ==> on va en 8 pour remettre le filament en auto si on n'a pas LE retour de VH ouverte, ça veut dire qu'on est passé en isolement ou en repompage*)
ELSIF	OP_RAH.Etape.6
		AND Timer_Reprise_Pompage.Q
		THEN
				OP_RAH.Etape.8 := TRUE;
				OP_RAH.Etape.6 := FALSE;

(*étape 7-8 ==> tempo de redémarrage - doit être courte, pusiqu'on ne fait que la remettre en auto, sans redémarrer le filament*)
ELSIF	OP_RAH.Etape.7
		AND TIMER_Restart_Jauge.Q
		THEN
				OP_RAH.ETAPE.8:=TRUE;
				OP_RAH.ETAPE.7:=FALSE;

(*étape 8-9 ==> envoi de mise en auto du filament réussi*)
ELSIF	OP_RAH.Etape.8
		AND NOT WRITE_CoE_BOOL.STATE_Busy
		AND NOT WRITE_CoE_BOOL.STATE_Error
		THEN
				OP_RAH.ETAPE.9:=TRUE;
				OP_RAH.ETAPE.8:=FALSE;

(*étape 8-12 ==> envoi de mise en auto du filament échoué*)
ELSIF	OP_RAH.Etape.8
		AND NOT WRITE_CoE_BOOL.STATE_Busy
		AND WRITE_CoE_BOOL.STATE_Error
		THEN
				OP_RAH.ETAPE.12:=TRUE;
				OP_RAH.ETAPE.8:=FALSE;

(*étape 9-10 ==> libre*)
ELSIF	OP_RAH.Etape.9
		THEN
				OP_RAH.ETAPE.10:=TRUE;
				OP_RAH.ETAPE.9:=FALSE;

(*étape 10-0 ==> libre*)
ELSIF	OP_RAH.Etape.10
		THEN
				OP_RAH.ETAPE.0:=TRUE;
				OP_RAH.ETAPE.10:=FALSE;

(*étape 12-0 ==> pb envoi de la commande*)
ELSIF	OP_RaH.Etape.12
		THEN
				OP_RaH.Etape.0 := TRUE;
				OP_RaH.Etape.12 := FALSE;

END_IF

OP_RAH.POST();
END_ACTION

END_FUNCTION_BLOCK

// ---- POUs/FONCTION DE BASE/WRITE_CoE_WORD.TcPOU
FUNCTION_BLOCK WRITE_CoE_WORD
(* Fonction standard AC d'écriture d'un paramètre CoE de type MOT (2 bytes) *)

(****************historique des versions*****************************)

(* Version 1-0 - AB - Version initiale - aff 8760*)
(* Codage selon exemple d'utilisation de  FB_EcCoESdoWrite dans InfoSystem *)
(*************************************************************************)

VAR_INPUT
	IN_NetId 		: T_AmsNetId; 				(* NetId of EtherCAT Master : on le trouve dans le .tsm, sur le device ethercat , onglet ethercat, champ NetId *)
	IN_SlaveAddr 	: UINT; 						(* Port Number of EtherCAT Slave *)
	IN_Index 		: WORD; 						(* CoE Object Index *)
	IN_SubIndex	 	: BYTE; 						(* Subindex of CoE Object *)
	IN_Value 		: WORD;						(* variable to be written to the CoE Object *)
	IN_ON		 	: BOOL;						(* rising edge starts writing to the CoE Object *)
END_VAR


VAR
	fbSdoWrite 	: FB_EcCoESdoWrite;
END_VAR

VAR_OUTPUT
	STATE_Busy:		BOOL;					(*en cours de traitement*)
	STATE_Error:	BOOL;					(* envoi raté si valeur à 1*)
	STATE_ErrId:	UDINT;					(* code erreur de l'échec de l'envoi*)
END_VAR

fbSdoWrite(
	sNetId 		:= IN_NetId,
	nSlaveAddr 	:= IN_SlaveAddr,
	nIndex 		:= IN_Index,
	nSubIndex 	:= IN_SubIndex,
	pSrcBuf 		:= ADR(IN_Value),
	cbBufLen 	:= SIZEOF(IN_Value),
	bExecute 	:= IN_ON
);

STATE_Busy := fbSdoWrite.bBusy;

IF NOT fbSdoWrite.bBusy THEN
	IN_ON := FALSE;
	IF NOT STATE_Error THEN
		(* write successful *)
		STATE_Error := FALSE;
		STATE_ErrId := 0;
	ELSE 
		(* write failed *)
		STATE_Error := fbSdoWrite.bError;
		STATE_ErrId := fbSdoWrite.nErrId;
	END_IF

	fbSdoWrite(bExecute := FALSE);
END_IF

END_FUNCTION_BLOCK

// ---- POUs/FONCTION DE BASE/WRITE_CoE_BOOL.TcPOU
FUNCTION_BLOCK WRITE_CoE_BOOL
(* Fonction standard AC d'écriture d'un paramètre CoE de type bool *)

(****************historique des versions*****************************)

(* Version 1-0 - AB - Version initiale - aff 8760*)
(* Codage selon exemple d'utilisation de  FB_EcCoESdoWrite dans InfoSystem *)
(*************************************************************************)

VAR_INPUT
	IN_NetId 		: T_AmsNetId; 				(* NetId of EtherCAT Master : on le trouve dans le .tsm, sur le device ethercat , onglet ethercat, champ NetId *)
	IN_SlaveAddr 	: UINT; 						(* Port Number of EtherCAT Slave *)
	IN_Index 		: WORD; 						(* CoE Object Index *)
	IN_SubIndex	 	: BYTE; 						(* Subindex of CoE Object *)
	IN_Value 		: BOOL;						(* variable to be written to the CoE Object *)
	IN_ON		 	: BOOL;						(* rising edge starts writing to the CoE Object *)
END_VAR


VAR
	fbSdoWrite 	: FB_EcCoESdoWrite;
	FD_Busy:	F_TRIG;				(*front descendant du state_busy pour etre sur de le voir passer*)
END_VAR

VAR_OUTPUT
	STATE_Busy:		BOOL;					(*en cours de traitement*)
	STATE_Error:		BOOL;					(* envoi raté si valeur à 1*)
	STATE_ErrId:			UDINT;					(* code erreur de l'échec de l'envoi*)

	toto : BOOL;
END_VAR

fbSdoWrite(
	sNetId 		:= IN_NetId,
	nSlaveAddr 	:= IN_SlaveAddr,
	nIndex 		:= IN_Index,
	nSubIndex 	:= IN_SubIndex,
	pSrcBuf 	:= ADR(IN_Value),
	cbBufLen 	:= SIZEOF(IN_Value),
	bExecute 	:= IN_ON
);

STATE_Busy := fbSdoWrite.bBusy;
FD_Busy(clk := STATE_Busy);

IF NOT fbSdoWrite.bBusy THEN
(*IF FD_Busy.Q THEN*)
	IN_ON := FALSE;
	IF NOT STATE_Error THEN
		(* write successful *)
		STATE_Error := FALSE;
		STATE_ErrId := 0;
	ELSE
		(* write failed *)
		STATE_Error := fbSdoWrite.bError;
		STATE_ErrId := fbSdoWrite.nErrId;
	END_IF

	fbSdoWrite(bExecute := FALSE);
END_IF

END_FUNCTION_BLOCK

// ---- POUs/Composant/POMPES/CRYO CTI/BLOCK_RS232_ONBOARD_V4.TcPOU
FUNCTION_BLOCK BLOCK_RS232_ONBOARD_V4
(* Communication RS232 - pour module On-Board Brooks *)
(*Gestion d'une seule pompe*)

(****************historique des versions*****************************)

(* Version 1-0 - HG - VERSION INIITIALE*)
(* Version 2-0 - LDS - 14136 - 04/2024 - Ajout parametrage cryo *)
(* Version 3-0 - LDS - 14136 - 07/2024 - Ajout gestion lecture information regen auto *)
(* Version 3-1 - LDS - 14624 - 21/03/2025 - Fusion des deux blocs avec déclaration conditionnel *)

(*************************************************************************)

VAR_INPUT
	CO_Etat:					BOOL;							(* Commande 1 = Marche de la pompe*)
	CO_Regen:					BOOL;							(* Demande de mise en régénération de la pompe *)
	CO_StopRegen:				BOOL;							(* Demande arrêt de la regeneration *)
	CO_Param_ParDefaut:			BOOL;							(* Demande paramétrage par defaut de regen cryo*)
	CO_states_regen:            BOOL;							(* Demande info regen lors d'un lancement auto*)
	
	CO_Ecriture:                BOOL;							(* Permet d'écrire les entré des parametres de la regen ds la pompe*)
	CO_Lecture:					BOOL;							(* Permet de lire les parametres de la regen enregistrer ds la pompe*)
	CO_RoughValve: 				BOOL;							(* Commande 1 = ouverture de la rough valve*)
	CO_PurgeValve:				BOOL;							(* Commande 1 = Marche de la purge valve*)
	CO_InfoPompe:				BOOL; 							(* demande Info de la Pompe *)
	CO_PumpTc:					BOOL; 							(* demande activation TC pump *)
	
	CO_Lecture_Relay:           BOOL;							(* permet de lire les relays(qd = true les infos des relais sont recupérées)*)
	CO_Envoie_Param_Relay:   	BOOL;							(* permet d'envoyer les parametres du relay*)
	CO_Param_usine_Relay:       BOOL;							(* parametrage par defaut des 2 relays *)
	
	CO_Forcage:					BOOL;							(* Permet de forcer sur une trame particuliere numero de trame dans ValeurForcageCptSend *)
	CONF_Forcage:				USINT;			(* Numero de la trame qui doit etre forcer avec le bool ForcageCptSend *)
	
	RESET:						BOOL;			(* Reset du driver*)
	OFF:						BOOL;			(* Désactivation du driver *)

	CO_ModeManu:				BOOL;			(* Passage en envoi manuel *)
	CO_EnvoiManu:				BOOL;			(* Commande d'envoi en mode manuel *)
	PRM_TrameManu:				STRING;			(* Contient la trame pour l'envoi manuel *)
	


	DEF_Port_com:				PRCDEF;			(* Defaut du port de communication rs232*)
	
    IN_COM			AT %I* :	PcComInData; 	//a mettre si liaison RS direct
    //IN_COM			AT %I* :	EL6inData22B;	//a mettre si liaison via carte EL6001
END_VAR
VAR_INPUT PERSISTENT
	(*Entité*)
	IsComponent:		BOOL;			(*entité : composant*)
	IdXML:				STRING;			(*nom entité : identifiant pour recherche dans dico*)
	TagXML:				UINT;			(*nom entité : identifiant pour recherche dans dico*)
	IdParent:			STRING;			(*MNEMO de l'appelant*)
	MNEMO:				STRING;			(*MNEMO de l'entité*)
	
	
	PRM_PowerFailRecovery:   USINT;
	PRM_PumpStartDelay:		 REAL;							(*parametres de la regen*)
	PRM_PumpRestartDelay:	 REAL;
	PRM_ExtendedPurgeTime:	 UINT;
	PRM_RepurgeCycles:	     USINT;
	PRM_RoughToPressure:	 USINT;
	PRM_ROR:	             USINT;
	PRM_RORCycles:	         USINT;
	PRM_StartUpTemperature:	 USINT;
	PRM_RoughValveInterlock: BOOL;
	PRM_RepurgeTime:	     REAL;
	PRM_1st_stage_control_temp: USINT:=65; 
												 			(*parametres des relais*)
	PRM_Relay:               USINT:=1;      (*num relais*)
	PRM_Action:				 USINT;	 	 (*commande*)
	PRM_Valeur:              UINT;		 (*valeur numerique associé a la commande*)
	PRM_ONOFF:               BOOL;		 (*Etat du relais*)
	PRM_Mode:				 BOOL;		 (*mode du relais*)
END_VAR
VAR_IN_OUT PERSISTENT

END_VAR 
VAR_OUTPUT
	REGEN_ERROR:                STRING;        			(* Donne l'erreur qui a stoppé la regen uniquement en anglais donc plus utilisé mais tjr fonctionnel*)
	STATE_Temperature:			ARRAY[0..1] OF REAL;	(* Donne la température de chaque étage d'une pompe *)
    STATE_Pressure:				REAL:=0.0;				(* Donne la pression "Thermocouple Gauge Pressure" *)
	STATE_Regen:				BOOL;			   	   	(* Donne l'etat de la regen *)
	Regen_completed:            BOOL;					(* Donne l'info si la regen a ete complete ou interrompu *)
	STEP_Regen:                 STRING;			 		(* Donne où en est la pompe dans le processus de regen*)
	STATE_Pompe:				BOOL;			 		(* Donne l'etat du moteur de la cryo *)
	STATE_Rough_valve: 			BOOL;					(*etat de la rough valve*)
	STATE_Purge_valve: 			BOOL;					(* etat de la vanne de purge*)
	STATE_Pump_TC: 				BOOL;					(* etat du pump TC*)
	Reponse_ModeManu:           STRING;					(* renvoie une chaine de caractere correspondant a la trame envoyé manuellement *)
	STATE_Tps_restant:          INT;					(* Donne le tps restant d'une étape de la regen *)
	STEP_REGEN_ID: 				UINT;					(* Donne l'étape de la regen en INT (utilisé pour les traduction) *)
	Pump_Serial_Number_affiche: STRING;    		        (* donne le numéro de serie de la pompe (complet) *)
	Number_Of_Complete_Regen:   UINT;					(* donne le nombre de cycle de regen completé *)
	Time_Since_Last_Regen:      UINT;					(* donne le tps depuis la dernière regen*)
	SoftwareRevisionLevel:      STRING;					(* donne la version du logiciel *)
	ElaspedTime:				UDINT;					(* donne le tps ecoulé*)
	ID_ERREUR_REGEN:            UINT:=1000;				(* donne l'ID de l'erreur (permet la traduction) *)
	NB_FAIL_PURGE_REPURGE:      UINT;					(* permet de  savoir le nombre d'echec de purge*)
	

    OUT_Com     AT %Q* : 	PcComOutData; 	//a mettre si liaison RS direct
    //OUT_Com		AT %Q* : 	EL6outData22B;	//a mettre si liaison via carte EL6001
	
	(*OUT_DTR_RTS 	AT %Q* : 		UINT;*)
	STATE_Ready:				BOOL;			(* Driver en fonctionnement *)
	STATE_NOK:					BOOL;			(* Driver en défaut *)
	
	VAR_Affichage :       		    STRING:='';		(*variable qui permette d'affiche des info supplémentaire sur l'étage de la regen*)
	VAR_Affichage_Commande_Relay:   UINT :=1000;		(*variable qui permet d'affiche la commande correspondant a la valeur numérique*)
	VAR_Affichage_Valeur_Relay:     STRING;			(*variable qui permet d'affiche la valeur actuelle enregistrer dans le relais (lié au champs de txt IHM*)
	TAB_Affichage_Etat_Relay:       ARRAY[1..2] OF BOOL;(*tableau permettant de stocker la valeur de l'état des 2 relais ON/OFF*)
	TAB_Affichage_Mode_relay:	    ARRAY[1..2] OF BOOL;(*tableau permettant de stocker la valeur du mode des 2 relais AUTO/MANU*)
	VAR_Affichage_ValeurTIME_Relay: STRING;			(*variable qui permet d'affiche la valeur du timer actuelle enregistrer dans le relais (lié au champs de txt IHM*)
	
	STATE_ROR_nb: 				 INT;				(*Nombre de cycle ROR*)
	LAST_ROR_Value:				 INT;				(*dernière valeur ROR*)
	VAR_Derniere_commande_Relay: STRING;			(*variable qui contient la dernière commande utilisé*)
	
	ID_COMBOBOX:                USINT;				(* ID de la combox permettant de le choix PowerFailRecovery*)
	ID_COMBOBOX_relay:          USINT;
	
	iCounter_Regen_lecture:     INT:=0;				(*compteur permettant de lire chaque parametre de la regen*)
END_VAR

VAR
	TIMER_Cadence: 				TON;			(*Timer cadencement communication*)
	TIMER_Demarrage: 			TON;			(*timer pour le démarrage et lorsqu'il arrete de communiquer*) 
	TIMER_Delay_Relay:          TON;			(*timer qui permet d'appliquer le délai lorqu'on repasse le relais en mode auto*) 
	TIMER_Delay_Relay2:         TON;			(*timer qui permet d'appliquer le délai lorqu'on change l'etat du relais (on/off)*)
	Var_lancement_timer_ONOFF: BOOL;			(* .IN du timer_delay_relay2 *)
 
	VAR_Cadence:				USINT;			(*Numéro de la trame en cours*)
	VAR_Mem_Cadence:			USINT;			(*Mémorisation numéro dela trame*)

	OUT_Send_Data:				SendString;		(*Fonction d'envoi*)
	OUT_Buffer: 				ComBuffer;		(*Buffer trame d'envoi *)

	IN_Receive_Data:			ReceiveString;	(*Fonction de réception*)
	IN_Buffer: 					ComBuffer;		(*Buffer trame de réception *)

	VAR_ClearBuffer: 			ClearComBuffer;	(*Fonction de RAZ buffer*)

	(* background communication with the COM port device *)
	VAR_COMportControl: 		SerialLineControl;
	VAR_COMportControlError: 	BOOL;
	VAR_COMportControlErrorID: 	ComError_t;
												(*ensembles des variables qui permettent de structurer les trames*)
	VAR_NB:						USINT;		 
	VAR_NB2:					USINT;
	VAR_BuffString:				STRING;
	VAR_TrameRetour:            STRING;
	VAR_STR1:					STRING[1];
	VAR_STR2:					STRING[1];
	VAR_ReceptionOk:			BOOL;
												(*ensemble des fronts montants/descendants pour la memorisation des commandes*)
	FM_Param: 					R_TRIG;				
	FM_On:						R_TRIG;
	FD_Off:						F_TRIG;
	FM_Regen:					R_TRIG;
	FM_StopRegen:				R_TRIG;
	FM_Ecriture:				R_TRIG;
	FM_Lecture:                 R_TRIG;
	FM_RoughValveOn:			R_TRIG;
	FM_RoughValveOff:			F_TRIG;
	FM_PurgeValveOn:            R_TRIG;
	FM_PurgeValveOff:           F_TRIG;
	FM_pump_TC_ON:				R_TRIG;
	FM_pump_TC_OFF:				F_TRIG;
	FM_EnvoieParamRelay:        R_TRIG;
	FM_InfoPompe  :             R_TRIG;
	FM_LectureRelay  :          R_TRIG;
	FM_ParamUsineRelay:         R_TRIG;
	FM_states_regen:            R_TRIG;
												(*ensemble des variables memorisation des commandes*)
	VAR_Mem_CO_Info_Pompe:     		BOOL;
	VAR_Mem_CO_RoughValve_on:  	 	BOOL;
	VAR_Mem_CO_RoughValve_off:  	BOOL;
	VAR_Mem_CO_PumpTC_on:  	 		BOOL;
	VAR_Mem_CO_PumpTC_off:  		BOOL;
	VAR_Mem_CO_PurgeValve_on:   	BOOL;
	VAR_Mem_CO_PurgeValve_off:  	BOOL;
	VAR_Mem_CO_Param_ParDefaut: 	BOOL;
	VAR_Mem_CO_On:					BOOL;
	VAR_Mem_CO_Off:					BOOL;
	VAR_Mem_CO_Regen:				BOOL;
	VAR_Mem_CO_StopRegen:      	    BOOL;
	VAR_Mem_CO_Ecriture:        	BOOL;
	VAR_Mem_CO_Lecture:         	BOOL;
	VAR_Reception_Parametre:    	BOOL := TRUE;
	VAR_Mem_Regen_Aborted:      	BOOL;
	VAR_Mem_CO_Lecture_Relay:      	BOOL;
	VAR_Mem_CO_Envoie_Param_Relay: 	BOOL;
	VAR_Mem_etape_Regen : 			BOOL;   (* variable qui permet de savoir si il faut lire les etapes de la regen*)
	VAR_Mem_CO_Param_usine_Relay:   BOOL;
	
	A_error: ComError_t;
	
	
	
	iCounter_ModeManu_lectureRegen:         INT:=0;
	iCounter_Regen_ecriture:                INT:=0;		(*compteur permettant d'affecter chaque parametre de la regen*)
	iCounter_Valeur_Num_Regen: 				INT:=0;		(*compteur permettant de demande les valeurs numériques de la regen (pour les étapes)*)
	iCounter_Info_Pompe: 					INT:=0;		(*compteur permettant de demande les infos de la pompe*)
	iCounter_Evitement_1ere_requete_regen:  INT:=0;
	iCounter_Param_Relay_lecture: 			INT:=0;
	
	VAR_Affichage1 :              STRING;			(*variables qui permettent de stocker des info supplémentaire sur l'étape de la regen (var concatenées)*)
	VAR_Affichage2 :              STRING;
	VAR_Affichage3 :              STRING;
	VAR_Affichage_ValeurUL_Relay: STRING;			(*var stocker la valeur UL du relais (concaténer dans une variable d'affichage total) *)
	VAR_Affichage_ValeurLL_Relay: STRING;			(*var stocker la valeur LL du relais (concaténer dans une variable d'affichage total) *)
	
	Pump_Serial_Number:	STRING;			            (* première partie du numéro de serie de la pompe *)
			
	STOP_LOAD:                   BOOL := FALSE;			(* Variables permettant de stopper la barre de chargement sur l'IHM*)
	VAR_Visibilite_valeur_relay: BOOL := FALSE;			(* Variables permettant de rendre invisible l'entre des valeur pour certaine commande dans les relays*)
	iCounter_Param_ParDefaut_Relay_lecture: INT;
	
	Message_alerte_invisible: BOOL:= TRUE;
	Message_alerte_invisible2: BOOL:= TRUE;
	Message_confirm_invisible: BOOL:= TRUE;
	Message_confirm_invisible_regen: BOOL:= TRUE;
	var_STRING: STRING(255);
	VAR_Demande_Erreur: BOOL;
END_VAR

(*Cadence :
Trame 1 : Demande état marche/arrêt - A?
Trame 2 : Demande état regen - O
Trame 3 : Demande si il y a eu des erreurs de regen  - e
Trame 6 : Demande température étage 1 - J
Trame 7 : Demande température étage 2 - K
Trame 5 : Demande pression - L
Trame 4 : Demande rought valve - D?
Trame 5 : Demande purge valve - E?
Trame 9 : Demande de regen d'une pompe / arret de regen - N1 / N0
Trame 10 : Demande de marche ou d'arrêt d'une pompe - A1 / A0
Trame 11 : Paramétrage regen P + [0 - 6,A,G][5 digit number]  ecriture
Trame 12 : Paramétrage regen P + [0 - 6,A,G][?]  lecture
Trame 13 : Demande étape dans la regen - O
Trame 14 : Demande d'ouverture de la rough valve - D0/D1
Trame 15 : Demande d'ouverture de la purge valve - E0/E1
Trame 16 : Demande info pompe
Trame 17 : Ecriture des parameres dans le relais
Trame 18 : Lecture des infos du relais (uniquement)
*)

(* Paramètre statique *)
IdXML							:=	'8';
TagXML							:=	2;

DEF_Port_com.IdXml				:=	'11';
DEF_Port_com.TagXml				:=	1;

(*Gestion PRM_Action impossible*)
IF PRM_Action = 9 OR PRM_Action = 14 THEN 
	PRM_Action := 0;
END_IF

IF PRM_Action =10 OR PRM_Action =11 OR PRM_Action =12 OR PRM_Action =13 OR PRM_Action =15 THEN
	VAR_Visibilite_valeur_relay:= TRUE;
ELSE
	VAR_Visibilite_valeur_relay:= FALSE;
END_IF

